LIN {X 0,Y 526.698,Z 428.469,A -85,B 0,C 180,E1 -4749.903,E2 -4749.903} C_VEL
LIN {X 0,Y 526.188,Z 442.456,A -85,B 0,C 180,E1 -4750.797,E2 -4750.797} C_VEL
LIN {X 0,Y 525.617,Z 456.418,A -85,B 0,C 180,E1 -4751.866,E2 -4751.866} C_VEL
LIN {X 0,Y 525.179,Z 468.801,A -85,B 0,C 180,E1 -4752.978,E2 -4752.978} C_VEL
LIN {X 0,Y 524.752,Z 481.132,A -85,B 0,C 180,E1 -4754.263,E2 -4754.263} C_VEL
LIN {X 0,Y 524.384,Z 492.437,A -85,B 0,C 180,E1 -4755.644,E2 -4755.644} C_VEL
LIN {X 0,Y 524.046,Z 503.255,A -85,B 0,C 180,E1 -4757.215,E2 -4757.215} C_VEL
LIN {X 0,Y 523.793,Z 512.276,A -85,B 0,C 180,E1 -4758.781,E2 -4758.781} C_VEL
LIN {X 0,Y 523.564,Z 519.801,A -85,B 0,C 180,E1 -4760.34,E2 -4760.34} C_VEL
LIN {X 0,Y 523.503,Z 526.021,A -85,B 0,C 180,E1 -4761.896,E2 -4761.896} C_VEL
LIN {X 0,Y 523.45,Z 531.029,A -85,B 0,C 180,E1 -4763.485,E2 -4763.485} C_VEL
LIN {X 0,Y 523.398,Z 533.892,A -85,B 0,C 180,E1 -4764.606,E2 -4764.606} C_VEL
LIN {X 0,Y 523.38,Z 536.906,A -85,B 0,C 180,E1 -4766.15,E2 -4766.15} C_VEL
LIN {X 0,Y 523.33,Z 538.868,A -85,B 0,C 180,E1 -4767.691,E2 -4767.691} C_VEL
LIN {X 0,Y 523.247,Z 539.833,A -85,B 0,C 180,E1 -4769.23,E2 -4769.23} C_VEL
LIN {X 0,Y 523.247,Z 539.832,A -85,B 0,C 180,E1 -4770.769,E2 -4770.769} C_VEL
LIN {X 0,Y 523.33,Z 538.868,A -85,B 0,C 180,E1 -4772.308,E2 -4772.308} C_VEL
LIN {X 0,Y 523.38,Z 536.906,A -85,B 0,C 180,E1 -4773.849,E2 -4773.849} C_VEL
LIN {X 0,Y 523.397,Z 533.906,A -85,B 0,C 180,E1 -4775.393,E2 -4775.393} C_VEL
LIN {X 0,Y 523.457,Z 529.853,A -85,B 0,C 180,E1 -4776.94,E2 -4776.94} C_VEL
LIN {X 0,Y 523.523,Z 524.622,A -85,B 0,C 180,E1 -4778.491,E2 -4778.491} C_VEL
LIN {X 0,Y 523.624,Z 518.224,A -85,B 0,C 180,E1 -4780.048,E2 -4780.048} C_VEL
LIN {X 0,Y 523.883,Z 510.045,A -85,B 0,C 180,E1 -4781.676,E2 -4781.676} C_VEL
LIN {X 0,Y 524.093,Z 501.032,A -85,B 0,C 180,E1 -4783.177,E2 -4783.177} C_VEL
LIN {X 0,Y 524.474,Z 491.393,A -85,B 0,C 180,E1 -4784.551,E2 -4784.551} C_VEL
LIN {X 0,Y 524.874,Z 480.123,A -85,B 0,C 180,E1 -4785.931,E2 -4785.931} C_VEL
LIN {X 0,Y 525.428,Z 466.759,A -85,B 0,C 180,E1 -4787.314,E2 -4787.314} C_VEL
LIN {X 0,Y 525.923,Z 454.174,A -85,B 0,C 180,E1 -4788.417,E2 -4788.417} C_VEL
LIN {X 0,Y 526.459,Z 439.758,A -85,B 0,C 180,E1 -4789.495,E2 -4789.495} C_VEL
LIN {X 0,Y 527.012,Z 425.551,A -85,B 0,C 180,E1 -4790.388,E2 -4790.388} C_VEL
LIN {X 0,Y 527.61,Z 410.217,A -85,B 0,C 180,E1 -4791.184,E2 -4791.184} C_VEL
LIN {X 0,Y 528.07,Z 394.743,A -85,B 0,C 180,E1 -4791.822,E2 -4791.822} C_VEL
LIN {X 0,Y 528.514,Z 378.995,A -85,B 0,C 180,E1 -4792.322,E2 -4792.322} C_VEL
LIN {X 0,Y 528.836,Z 362.769,A -85,B 0,C 180,E1 -4792.694,E2 -4792.694} C_VEL
LIN {X 0,Y 529.26,Z 309.626,A -85,B 0,C 180,E1 -4793.476,E2 -4793.476} C_VEL
LIN {X 0,Y 530.388,Z 201.86,A -85,B 0,C 180,E1 -4795.062,E2 -4795.062} C_VEL
LIN {X 0,Y 530.606,Z 171.21,A -85,B 0,C 180,E1 -4795.535,E2 -4795.535} C_VEL
LIN {X 0,Y 528.283,Z 155.627,A -85,B 0,C 180,E1 -4795.933,E2 -4795.933} C_VEL
LIN {X 0,Y 529.372,Z 120.749,A -85,B 0,C 180,E1 -4798.908,E2 -4798.908} C_VEL
LIN {X 0,Y 529.593,Z 109.375,A -85,B 0,C 180,E1 -4799.898,E2 -4799.898} C_VEL
LIN {X 0,Y 523.945,Z 91.535,A -85,B 0,C 180,E1 -4801.852,E2 -4801.852} C_VEL
LIN {X 0,Y 523.935,Z 91.535,A -85,B 0,C 180,E1 -4804.289,E2 -4804.289} C_VEL
LIN {X 0,Y 523.903,Z 91.537,A -85,B 0,C 180,E1 -4807.132,E2 -4807.132} C_VEL
LIN {X 0,Y 523.933,Z 91.535,A -85,B 0,C 180,E1 -4810.129,E2 -4810.129} C_VEL
LIN {X 0,Y 523.935,Z 91.538,A -85,B 0,C 180,E1 -4812.459,E2 -4812.459} C_VEL
LIN {X 0,Y 523.951,Z 91.528,A -85,B 0,C 180,E1 -4815.308,E2 -4815.308} C_VEL
LIN {X 0,Y 523.954,Z 91.53,A -85,B 0,C 180,E1 -4818.689,E2 -4818.689} C_VEL
LIN {X 0,Y 523.913,Z 91.535,A -85,B 0,C 180,E1 -4821.898,E2 -4821.898} C_VEL
LIN {X 0,Y 523.934,Z 91.53,A -85,B 0,C 180,E1 -4824.909,E2 -4824.909} C_VEL
LIN {X 0,Y 523.934,Z 91.531,A -85,B 0,C 180,E1 -4827.679,E2 -4827.679} C_VEL
LIN {X 0,Y 523.956,Z 91.528,A -85,B 0,C 180,E1 -4830.675,E2 -4830.675} C_VEL
LIN {X 0,Y 523.97,Z 91.528,A -85,B 0,C 180,E1 -4833.728,E2 -4833.728} C_VEL
LIN {X 0,Y 523.932,Z 91.535,A -85,B 0,C 180,E1 -4836.271,E2 -4836.271} C_VEL
LIN {X 0,Y 523.941,Z 91.528,A -85,B 0,C 180,E1 -4838.767,E2 -4838.767} C_VEL
LIN {X 0,Y 523.948,Z 91.528,A -85,B 0,C 180,E1 -4841.221,E2 -4841.221} C_VEL
LIN {X 0,Y 523.933,Z 91.534,A -85,B 0,C 180,E1 -4843.639,E2 -4843.639} C_VEL
LIN {X 0,Y 523.937,Z 91.535,A -85,B 0,C 180,E1 -4846.028,E2 -4846.028} C_VEL
LIN {X 0,Y 524.01,Z 91.521,A -85,B 0,C 180,E1 -4848.394,E2 -4848.394} C_VEL
LIN {X 0,Y 523.999,Z 91.526,A -85,B 0,C 180,E1 -4851.516,E2 -4851.516} C_VEL
LIN {X 0,Y 524.078,Z 91.511,A -85,B 0,C 180,E1 -4854.614,E2 -4854.614} C_VEL
LIN {X 0,Y 524.107,Z 91.516,A -85,B 0,C 180,E1 -4857.695,E2 -4857.695} C_VEL
LIN {X 0,Y 524.119,Z 91.506,A -85,B 0,C 180,E1 -4860.768,E2 -4860.768} C_VEL
LIN {X 0,Y 524.069,Z 91.514,A -85,B 0,C 180,E1 -4863.075,E2 -4863.075} C_VEL
LIN {X 0,Y 524.042,Z 91.517,A -85,B 0,C 180,E1 -4866.159,E2 -4866.159} C_VEL
LIN {X 0,Y 523.993,Z 91.527,A -85,B 0,C 180,E1 -4869.262,E2 -4869.262} C_VEL
LIN {X 0,Y 523.999,Z 91.525,A -85,B 0,C 180,E1 -4871.74,E2 -4871.74} C_VEL
LIN {X 0,Y 523.989,Z 91.526,A -85,B 0,C 180,E1 -4875.053,E2 -4875.053} C_VEL
LIN {X 0,Y 523.96,Z 91.527,A -85,B 0,C 180,E1 -4877.969,E2 -4877.969} C_VEL
LIN {X 0,Y 523.968,Z 91.525,A -85,B 0,C 180,E1 -4880.41,E2 -4880.41} C_VEL
LIN {X 0,Y 523.913,Z 91.536,A -85,B 0,C 180,E1 -4882.893,E2 -4882.893} C_VEL
LIN {X 0,Y 523.949,Z 91.532,A -85,B 0,C 180,E1 -4885.419,E2 -4885.419} C_VEL
LIN {X 0,Y 523.965,Z 91.525,A -85,B 0,C 180,E1 -4887.999,E2 -4887.999} C_VEL
LIN {X 0,Y 523.943,Z 91.533,A -85,B 0,C 180,E1 -4890.856,E2 -4890.856} C_VEL
LIN {X 0,Y 523.958,Z 91.527,A -85,B 0,C 180,E1 -4893.735,E2 -4893.735} C_VEL
LIN {X 0,Y 523.919,Z 91.532,A -85,B 0,C 180,E1 -4896.405,E2 -4896.405} C_VEL
LIN {X 0,Y 523.921,Z 91.537,A -85,B 0,C 180,E1 -4899.085,E2 -4899.085} C_VEL
LIN {X 0,Y 523.953,Z 91.527,A -85,B 0,C 180,E1 -4902.119,E2 -4902.119} C_VEL
LIN {X 0,Y 523.953,Z 91.529,A -85,B 0,C 180,E1 -4905.309,E2 -4905.309} C_VEL
LIN {X 0,Y 523.92,Z 91.538,A -85,B 0,C 180,E1 -4906.914,E2 -4906.914} C_VEL
LIN {X 0,Y 523.253,Z 91.616,A -85,B 0,C 180,E1 -4907.555,E2 -4907.555} C_VEL
LIN {X 0,Y 520.408,Z 91.974,A -85,B 0,C 180,E1 -4908.597,E2 -4908.597} C_VEL
LIN {X 0,Y 518.002,Z 92.271,A -85,B 0,C 180,E1 -4909.436,E2 -4909.436} C_VEL
LIN {X 0,Y 516.965,Z 92.399,A -85,B 0,C 180,E1 -4910.083,E2 -4910.083} C_VEL
LIN {X 0,Y 516.879,Z 92.41,A -85,B 0,C 180,E1 -4910.303,E2 -4910.303} C_VEL
LIN {X 0,Y 516.874,Z 92.409,A -85,B 0,C 180,E1 -4913.344,E2 -4913.344} C_VEL
LIN {X 0,Y 516.905,Z 92.406,A -85,B 0,C 180,E1 -4916.121,E2 -4916.121} C_VEL
LIN {X 0,Y 516.889,Z 92.411,A -85,B 0,C 180,E1 -4918.936,E2 -4918.936} C_VEL
LIN {X 0,Y 516.917,Z 92.403,A -85,B 0,C 180,E1 -4921.585,E2 -4921.585} C_VEL
LIN {X 0,Y 516.93,Z 92.406,A -85,B 0,C 180,E1 -4924.212,E2 -4924.212} C_VEL
LIN {X 0,Y 516.87,Z 92.413,A -85,B 0,C 180,E1 -4926.777,E2 -4926.777} C_VEL
LIN {X 0,Y 516.938,Z 92.401,A -85,B 0,C 180,E1 -4929.732,E2 -4929.732} C_VEL
LIN {X 0,Y 516.928,Z 92.407,A -85,B 0,C 180,E1 -4932.597,E2 -4932.597} C_VEL
LIN {X 0,Y 516.942,Z 92.401,A -85,B 0,C 180,E1 -4935.031,E2 -4935.031} C_VEL
LIN {X 0,Y 516.966,Z 92.406,A -85,B 0,C 180,E1 -4938.234,E2 -4938.234} C_VEL
LIN {X 0,Y 516.968,Z 92.397,A -85,B 0,C 180,E1 -4941.4,E2 -4941.4} C_VEL
LIN {X 0,Y 517.011,Z 92.395,A -85,B 0,C 180,E1 -4943.757,E2 -4943.757} C_VEL
LIN {X 0,Y 517.085,Z 92.385,A -85,B 0,C 180,E1 -4947.664,E2 -4947.664} C_VEL
LIN {X 0,Y 517.094,Z 92.382,A -85,B 0,C 180,E1 -4950.779,E2 -4950.779} C_VEL
LIN {X 0,Y 517.012,Z 92.391,A -85,B 0,C 180,E1 -4953.117,E2 -4953.117} C_VEL
LIN {X 0,Y 517.011,Z 92.396,A -85,B 0,C 180,E1 -4956.244,E2 -4956.244} C_VEL
LIN {X 0,Y 516.953,Z 92.401,A -85,B 0,C 180,E1 -4959.39,E2 -4959.39} C_VEL
LIN {X 0,Y 516.954,Z 92.407,A -85,B 0,C 180,E1 -4961.808,E2 -4961.808} C_VEL
LIN {X 0,Y 516.946,Z 92.4,A -85,B 0,C 180,E1 -4965.147,E2 -4965.147} C_VEL
LIN {X 0,Y 516.927,Z 92.404,A -85,B 0,C 180,E1 -4968.223,E2 -4968.223} C_VEL
LIN {X 0,Y 516.915,Z 92.403,A -85,B 0,C 180,E1 -4970.702,E2 -4970.702} C_VEL
LIN {X 0,Y 516.894,Z 92.409,A -85,B 0,C 180,E1 -4974.073,E2 -4974.073} C_VEL
LIN {X 0,Y 516.928,Z 92.402,A -85,B 0,C 180,E1 -4976.658,E2 -4976.658} C_VEL
LIN {X 0,Y 516.913,Z 92.412,A -85,B 0,C 180,E1 -4979.524,E2 -4979.524} C_VEL
LIN {X 0,Y 516.9,Z 92.405,A -85,B 0,C 180,E1 -4982.544,E2 -4982.544} C_VEL
LIN {X 0,Y 516.869,Z 92.416,A -85,B 0,C 180,E1 -4985.33,E2 -4985.33} C_VEL
LIN {X 0,Y 516.882,Z 92.409,A -85,B 0,C 180,E1 -4987.943,E2 -4987.943} C_VEL
LIN {X 0,Y 516.886,Z 92.408,A -85,B 0,C 180,E1 -4990.742,E2 -4990.742} C_VEL
LIN {X 0,Y 516.886,Z 92.409,A -85,B 0,C 180,E1 -4992.832,E2 -4992.832} C_VEL
LIN {X 0,Y 516.926,Z 92.407,A -85,B 0,C 180,E1 -4995.01,E2 -4995.01} C_VEL
LIN {X 0,Y 516.916,Z 92.403,A -85,B 0,C 180,E1 -4998.399,E2 -4998.399} C_VEL
LIN {X 0,Y 516.884,Z 92.414,A -85,B 0,C 180,E1 -5001.284,E2 -5001.284} C_VEL
LIN {X 0,Y 516.88,Z 92.409,A -85,B 0,C 180,E1 -5004.22,E2 -5004.22} C_VEL
LIN {X 0,Y 516.898,Z 92.414,A -85,B 0,C 180,E1 -5007.053,E2 -5007.053} C_VEL
LIN {X 0,Y 516.896,Z 92.409,A -85,B 0,C 180,E1 -5009.797,E2 -5009.797} C_VEL
LIN {X 0,Y 516.93,Z 92.408,A -85,B 0,C 180,E1 -5012.467,E2 -5012.467} C_VEL
LIN {X 0,Y 516.94,Z 92.407,A -85,B 0,C 180,E1 -5013.709,E2 -5013.709} C_VEL
LIN {X 0,Y 517.988,Z 95.336,A -85,B 0,C 180,E1 -5013.83,E2 -5013.83} C_VEL
LIN {X 0,Y 524.276,Z 108.483,A -85,B 0,C 180,E1 -5014.383,E2 -5014.383} C_VEL
LIN {X 0,Y 522.69,Z 254.21,A -85,B 0,C 180,E1 -5016.605,E2 -5016.605} C_VEL
LIN {X 0,Y 522.29,Z 290.172,A -85,B 0,C 180,E1 -5017.162,E2 -5017.162} C_VEL
LIN {X 0,Y 521.965,Z 307.306,A -85,B 0,C 180,E1 -5017.591,E2 -5017.591} C_VEL
LIN {X 0,Y 521.509,Z 323.109,A -85,B 0,C 180,E1 -5018.144,E2 -5018.144} C_VEL
LIN {X 0,Y 521.037,Z 338.718,A -85,B 0,C 180,E1 -5018.85,E2 -5018.85} C_VEL
LIN {X 0,Y 520.492,Z 353.18,A -85,B 0,C 180,E1 -5019.654,E2 -5019.654} C_VEL
LIN {X 0,Y 519.849,Z 368.084,A -85,B 0,C 180,E1 -5020.657,E2 -5020.657} C_VEL
LIN {X 0,Y 519.233,Z 381.509,A -85,B 0,C 180,E1 -5021.744,E2 -5021.744} C_VEL
LIN {X 0,Y 518.651,Z 393.241,A -85,B 0,C 180,E1 -5022.859,E2 -5022.859} C_VEL
LIN {X 0,Y 518.193,Z 404.191,A -85,B 0,C 180,E1 -5024.059,E2 -5024.059} C_VEL
LIN {X 0,Y 517.695,Z 415.067,A -85,B 0,C 180,E1 -5025.455,E2 -5025.455} C_VEL
LIN {X 0,Y 517.26,Z 425.524,A -85,B 0,C 180,E1 -5027.045,E2 -5027.045} C_VEL
LIN {X 0,Y 516.92,Z 434.225,A -85,B 0,C 180,E1 -5028.63,E2 -5028.63} C_VEL
LIN {X 0,Y 516.636,Z 441.519,A -85,B 0,C 180,E1 -5030.21,E2 -5030.21} C_VEL
LIN {X 0,Y 516.517,Z 447.491,A -85,B 0,C 180,E1 -5031.786,E2 -5031.786} C_VEL
LIN {X 0,Y 516.437,Z 452.437,A -85,B 0,C 180,E1 -5033.431,E2 -5033.431} C_VEL
LIN {X 0,Y 516.334,Z 455.124,A -85,B 0,C 180,E1 -5034.533,E2 -5034.533} C_VEL
LIN {X 0,Y 516.327,Z 458.021,A -85,B 0,C 180,E1 -5036.097,E2 -5036.097} C_VEL
LIN {X 0,Y 516.255,Z 459.965,A -85,B 0,C 180,E1 -5037.659,E2 -5037.659} C_VEL
LIN {X 0,Y 516.186,Z 460.93,A -85,B 0,C 180,E1 -5039.22,E2 -5039.22} C_VEL
LIN {X 0,Y 516.189,Z 460.981,A -85,B 0,C 180,E1 -5040.78,E2 -5040.78} C_VEL
LIN {X 0,Y 516.257,Z 460.095,A -85,B 0,C 180,E1 -5042.341,E2 -5042.341} C_VEL
LIN {X 0,Y 516.341,Z 458.242,A -85,B 0,C 180,E1 -5043.902,E2 -5043.902} C_VEL
LIN {X 0,Y 516.338,Z 455.456,A -85,B 0,C 180,E1 -5045.467,E2 -5045.467} C_VEL
LIN {X 0,Y 516.476,Z 451.597,A -85,B 0,C 180,E1 -5047.034,E2 -5047.034} C_VEL
LIN {X 0,Y 516.525,Z 446.628,A -85,B 0,C 180,E1 -5048.608,E2 -5048.608} C_VEL
LIN {X 0,Y 516.701,Z 440.491,A -85,B 0,C 180,E1 -5050.185,E2 -5050.185} C_VEL
LIN {X 0,Y 516.99,Z 432.998,A -85,B 0,C 180,E1 -5051.766,E2 -5051.766} C_VEL
LIN {X 0,Y 517.368,Z 423.951,A -85,B 0,C 180,E1 -5053.352,E2 -5053.352} C_VEL
LIN {X 0,Y 517.764,Z 414.573,A -85,B 0,C 180,E1 -5054.744,E2 -5054.744} C_VEL
LIN {X 0,Y 518.272,Z 403.549,A -85,B 0,C 180,E1 -5056.14,E2 -5056.14} C_VEL
LIN {X 0,Y 518.798,Z 391.418,A -85,B 0,C 180,E1 -5057.441,E2 -5057.441} C_VEL
LIN {X 0,Y 519.406,Z 378.461,A -85,B 0,C 180,E1 -5058.61,E2 -5058.61} C_VEL
LIN {X 0,Y 519.915,Z 364.877,A -85,B 0,C 180,E1 -5059.648,E2 -5059.648} C_VEL
LIN {X 0,Y 520.439,Z 350.731,A -85,B 0,C 180,E1 -5060.555,E2 -5060.555} C_VEL
LIN {X 0,Y 521.023,Z 335.381,A -85,B 0,C 180,E1 -5061.358,E2 -5061.358} C_VEL
LIN {X 0,Y 521.419,Z 319.929,A -85,B 0,C 180,E1 -5062.001,E2 -5062.001} C_VEL
LIN {X 0,Y 521.748,Z 303.332,A -85,B 0,C 180,E1 -5062.523,E2 -5062.523} C_VEL
LIN {X 0,Y 521.951,Z 287.036,A -85,B 0,C 180,E1 -5062.88,E2 -5062.88} C_VEL
LIN {X 0,Y 523.479,Z 165.935,A -85,B 0,C 180,E1 -5064.773,E2 -5064.773} C_VEL
LIN {X 0,Y 524.468,Z 108.668,A -85,B 0,C 180,E1 -5065.737,E2 -5065.737} C_VEL
LIN {X 0,Y 518.182,Z 95.78,A -85,B 0,C 180,E1 -5066.361,E2 -5066.361} C_VEL
LIN {X 0,Y 516.963,Z 93.096,A -85,B 0,C 180,E1 -5066.487,E2 -5066.487} C_VEL
LIN {X 0,Y 516.837,Z 92.42,A -85,B 0,C 180,E1 -5066.521,E2 -5066.521} C_VEL
LIN {X 0,Y 516.881,Z 92.414,A -85,B 0,C 180,E1 -5069.517,E2 -5069.517} C_VEL
LIN {X 0,Y 516.893,Z 92.415,A -85,B 0,C 180,E1 -5072.542,E2 -5072.542} C_VEL
LIN {X 0,Y 516.865,Z 92.414,A -85,B 0,C 180,E1 -5075.329,E2 -5075.329} C_VEL
LIN {X 0,Y 516.879,Z 92.414,A -85,B 0,C 180,E1 -5077.942,E2 -5077.942} C_VEL
LIN {X 0,Y 516.884,Z 92.413,A -85,B 0,C 180,E1 -5080.741,E2 -5080.741} C_VEL
LIN {X 0,Y 516.884,Z 92.412,A -85,B 0,C 180,E1 -5082.831,E2 -5082.831} C_VEL
LIN {X 0,Y 516.897,Z 92.409,A -85,B 0,C 180,E1 -5085.007,E2 -5085.007} C_VEL
LIN {X 0,Y 516.915,Z 92.41,A -85,B 0,C 180,E1 -5088.398,E2 -5088.398} C_VEL
LIN {X 0,Y 516.882,Z 92.414,A -85,B 0,C 180,E1 -5091.284,E2 -5091.284} C_VEL
LIN {X 0,Y 516.872,Z 92.417,A -85,B 0,C 180,E1 -5094.219,E2 -5094.219} C_VEL
LIN {X 0,Y 516.897,Z 92.418,A -85,B 0,C 180,E1 -5097.053,E2 -5097.053} C_VEL
LIN {X 0,Y 516.957,Z 92.588,A -85,B 0,C 180,E1 -5097.98,E2 -5097.98} C_VEL
LIN {X 0,Y 521.725,Z 108.054,A -85,B 0,C 180,E1 -5099.788,E2 -5099.788} C_VEL
LIN {X 0,Y 522.518,Z 111.509,A -85,B 0,C 180,E1 -5100.154,E2 -5100.154} C_VEL
LIN {X 0,Y 521.372,Z 141.954,A -85,B 0,C 180,E1 -5102.831,E2 -5102.831} C_VEL
LIN {X 0,Y 521.076,Z 151.687,A -85,B 0,C 180,E1 -5103.668,E2 -5103.668} C_VEL
LIN {X 0,Y 524.053,Z 173.701,A -85,B 0,C 180,E1 -5104.228,E2 -5104.228} C_VEL
LIN {X 0,Y 522.395,Z 292.457,A -85,B 0,C 180,E1 -5106.117,E2 -5106.117} C_VEL
LIN {X 0,Y 521.708,Z 362.986,A -85,B 0,C 180,E1 -5107.187,E2 -5107.187} C_VEL
LIN {X 0,Y 521.337,Z 380.565,A -85,B 0,C 180,E1 -5107.614,E2 -5107.614} C_VEL
LIN {X 0,Y 520.88,Z 396.793,A -85,B 0,C 180,E1 -5108.167,E2 -5108.167} C_VEL
LIN {X 0,Y 520.346,Z 412.264,A -85,B 0,C 180,E1 -5108.842,E2 -5108.842} C_VEL
LIN {X 0,Y 519.81,Z 426.912,A -85,B 0,C 180,E1 -5109.625,E2 -5109.625} C_VEL
LIN {X 0,Y 519.269,Z 441.013,A -85,B 0,C 180,E1 -5110.531,E2 -5110.531} C_VEL
LIN {X 0,Y 518.675,Z 455.327,A -85,B 0,C 180,E1 -5111.63,E2 -5111.63} C_VEL
LIN {X 0,Y 518.168,Z 468.684,A -85,B 0,C 180,E1 -5112.842,E2 -5112.842} C_VEL
LIN {X 0,Y 517.762,Z 480.106,A -85,B 0,C 180,E1 -5114.045,E2 -5114.045} C_VEL
LIN {X 0,Y 517.368,Z 491.488,A -85,B 0,C 180,E1 -5115.445,E2 -5115.445} C_VEL
LIN {X 0,Y 516.952,Z 502.384,A -85,B 0,C 180,E1 -5117.037,E2 -5117.037} C_VEL
LIN {X 0,Y 516.79,Z 509.654,A -85,B 0,C 180,E1 -5118.279,E2 -5118.279} C_VEL
LIN {X 0,Y 516.559,Z 517.352,A -85,B 0,C 180,E1 -5119.812,E2 -5119.812} C_VEL
LIN {X 0,Y 516.453,Z 523.852,A -85,B 0,C 180,E1 -5121.391,E2 -5121.391} C_VEL
LIN {X 0,Y 516.377,Z 529.177,A -85,B 0,C 180,E1 -5122.964,E2 -5122.964} C_VEL
LIN {X 0,Y 516.327,Z 533.277,A -85,B 0,C 180,E1 -5124.532,E2 -5124.532} C_VEL
LIN {X 0,Y 516.305,Z 536.329,A -85,B 0,C 180,E1 -5126.097,E2 -5126.097} C_VEL
LIN {X 0,Y 516.256,Z 538.32,A -85,B 0,C 180,E1 -5127.659,E2 -5127.659} C_VEL
LIN {X 0,Y 516.166,Z 539.314,A -85,B 0,C 180,E1 -5129.219,E2 -5129.219} C_VEL
LIN {X 0,Y 516.166,Z 539.319,A -85,B 0,C 180,E1 -5130.78,E2 -5130.78} C_VEL
LIN {X 0,Y 516.256,Z 538.349,A -85,B 0,C 180,E1 -5132.34,E2 -5132.34} C_VEL
LIN {X 0,Y 516.305,Z 536.374,A -85,B 0,C 180,E1 -5133.902,E2 -5133.902} C_VEL
LIN {X 0,Y 516.326,Z 533.364,A -85,B 0,C 180,E1 -5135.467,E2 -5135.467} C_VEL
LIN {X 0,Y 516.376,Z 529.3,A -85,B 0,C 180,E1 -5137.035,E2 -5137.035} C_VEL
LIN {X 0,Y 516.455,Z 524.047,A -85,B 0,C 180,E1 -5138.608,E2 -5138.608} C_VEL
LIN {X 0,Y 516.561,Z 517.619,A -85,B 0,C 180,E1 -5140.187,E2 -5140.187} C_VEL
LIN {X 0,Y 516.801,Z 509.778,A -85,B 0,C 180,E1 -5141.77,E2 -5141.77} C_VEL
LIN {X 0,Y 517.091,Z 500.371,A -85,B 0,C 180,E1 -5143.359,E2 -5143.359} C_VEL
LIN {X 0,Y 517.464,Z 489.152,A -85,B 0,C 180,E1 -5144.954,E2 -5144.954} C_VEL
LIN {X 0,Y 517.952,Z 477.535,A -85,B 0,C 180,E1 -5146.352,E2 -5146.352} C_VEL
LIN {X 0,Y 518.521,Z 464.876,A -85,B 0,C 180,E1 -5147.653,E2 -5147.653} C_VEL
LIN {X 0,Y 519.066,Z 451.613,A -85,B 0,C 180,E1 -5148.814,E2 -5148.814} C_VEL
LIN {X 0,Y 519.692,Z 437.359,A -85,B 0,C 180,E1 -5149.863,E2 -5149.863} C_VEL
LIN {X 0,Y 520.307,Z 422.946,A -85,B 0,C 180,E1 -5150.752,E2 -5150.752} C_VEL
LIN {X 0,Y 520.9,Z 407.287,A -85,B 0,C 180,E1 -5151.55,E2 -5151.55} C_VEL
LIN {X 0,Y 521.448,Z 392.036,A -85,B 0,C 180,E1 -5152.171,E2 -5152.171} C_VEL
LIN {X 0,Y 521.856,Z 375.621,A -85,B 0,C 180,E1 -5152.674,E2 -5152.674} C_VEL
LIN {X 0,Y 522.216,Z 359.174,A -85,B 0,C 180,E1 -5153.022,E2 -5153.022} C_VEL
LIN {X 0,Y 523.526,Z 237.483,A -85,B 0,C 180,E1 -5154.856,E2 -5154.856} C_VEL
LIN {X 0,Y 524.19,Z 172.24,A -85,B 0,C 180,E1 -5155.847,E2 -5155.847} C_VEL
LIN {X 0,Y 521.619,Z 155.534,A -85,B 0,C 180,E1 -5156.263,E2 -5156.263} C_VEL
LIN {X 0,Y 522.793,Z 121.957,A -85,B 0,C 180,E1 -5159.163,E2 -5159.163} C_VEL
LIN {X 0,Y 523.145,Z 112.783,A -85,B 0,C 180,E1 -5159.964,E2 -5159.964} C_VEL
LIN {X 0,Y 519.785,Z 101.473,A -85,B 0,C 180,E1 -5161.186,E2 -5161.186} C_VEL
LIN {X 0,Y 516.919,Z 92.411,A -85,B 0,C 180,E1 -5162.201,E2 -5162.201} C_VEL
LIN {X 0,Y 516.883,Z 92.415,A -85,B 0,C 180,E1 -5164.824,E2 -5164.824} C_VEL
LIN {X 0,Y 516.876,Z 92.412,A -85,B 0,C 180,E1 -5167.943,E2 -5167.943} C_VEL
LIN {X 0,Y 516.88,Z 92.415,A -85,B 0,C 180,E1 -5170.741,E2 -5170.741} C_VEL
LIN {X 0,Y 516.9,Z 92.41,A -85,B 0,C 180,E1 -5172.829,E2 -5172.829} C_VEL
LIN {X 0,Y 516.918,Z 92.406,A -85,B 0,C 180,E1 -5175.01,E2 -5175.01} C_VEL
LIN {X 0,Y 516.91,Z 92.412,A -85,B 0,C 180,E1 -5178.398,E2 -5178.398} C_VEL
LIN {X 0,Y 516.879,Z 92.408,A -85,B 0,C 180,E1 -5181.284,E2 -5181.284} C_VEL
LIN {X 0,Y 516.886,Z 92.416,A -85,B 0,C 180,E1 -5184.221,E2 -5184.221} C_VEL
LIN {X 0,Y 516.892,Z 92.406,A -85,B 0,C 180,E1 -5187.053,E2 -5187.053} C_VEL
LIN {X 0,Y 516.895,Z 92.409,A -85,B 0,C 180,E1 -5189.797,E2 -5189.797} C_VEL
LIN {X 0,Y 516.923,Z 92.406,A -85,B 0,C 180,E1 -5192.467,E2 -5192.467} C_VEL
LIN {X 0,Y 516.906,Z 92.404,A -85,B 0,C 180,E1 -5195.072,E2 -5195.072} C_VEL
LIN {X 0,Y 516.865,Z 92.413,A -85,B 0,C 180,E1 -5197.622,E2 -5197.622} C_VEL
LIN {X 0,Y 516.928,Z 92.408,A -85,B 0,C 180,E1 -5200.13,E2 -5200.13} C_VEL
LIN {X 0,Y 516.925,Z 92.403,A -85,B 0,C 180,E1 -5202.596,E2 -5202.596} C_VEL
LIN {X 0,Y 516.938,Z 92.4,A -85,B 0,C 180,E1 -5205.03,E2 -5205.03} C_VEL
LIN {X 0,Y 517,Z 92.396,A -85,B 0,C 180,E1 -5208.235,E2 -5208.235} C_VEL
LIN {X 0,Y 516.964,Z 92.401,A -85,B 0,C 180,E1 -5211.4,E2 -5211.4} C_VEL
LIN {X 0,Y 517.006,Z 92.401,A -85,B 0,C 180,E1 -5213.757,E2 -5213.757} C_VEL
LIN {X 0,Y 517.079,Z 92.392,A -85,B 0,C 180,E1 -5217.663,E2 -5217.663} C_VEL
LIN {X 0,Y 517.089,Z 92.382,A -85,B 0,C 180,E1 -5220.779,E2 -5220.779} C_VEL
LIN {X 0,Y 517.01,Z 92.394,A -85,B 0,C 180,E1 -5223.117,E2 -5223.117} C_VEL
LIN {X 0,Y 517.006,Z 92.393,A -85,B 0,C 180,E1 -5226.243,E2 -5226.243} C_VEL
LIN {X 0,Y 516.947,Z 92.407,A -85,B 0,C 180,E1 -5229.389,E2 -5229.389} C_VEL
LIN {X 0,Y 516.948,Z 92.403,A -85,B 0,C 180,E1 -5231.807,E2 -5231.807} C_VEL
LIN {X 0,Y 516.94,Z 92.406,A -85,B 0,C 180,E1 -5235.147,E2 -5235.147} C_VEL
LIN {X 0,Y 516.922,Z 92.402,A -85,B 0,C 180,E1 -5238.222,E2 -5238.222} C_VEL
LIN {X 0,Y 516.908,Z 92.406,A -85,B 0,C 180,E1 -5240.702,E2 -5240.702} C_VEL
LIN {X 0,Y 516.908,Z 92.404,A -85,B 0,C 180,E1 -5244.072,E2 -5244.072} C_VEL
LIN {X 0,Y 516.922,Z 92.405,A -85,B 0,C 180,E1 -5246.658,E2 -5246.658} C_VEL
LIN {X 0,Y 516.907,Z 92.407,A -85,B 0,C 180,E1 -5249.524,E2 -5249.524} C_VEL
LIN {X 0,Y 516.897,Z 92.408,A -85,B 0,C 180,E1 -5252.545,E2 -5252.545} C_VEL
LIN {X 0,Y 516.879,Z 92.412,A -85,B 0,C 180,E1 -5255.333,E2 -5255.333} C_VEL
LIN {X 0,Y 516.878,Z 92.408,A -85,B 0,C 180,E1 -5257.944,E2 -5257.944} C_VEL
LIN {X 0,Y 516.882,Z 92.414,A -85,B 0,C 180,E1 -5260.742,E2 -5260.742} C_VEL
LIN {X 0,Y 516.9,Z 92.413,A -85,B 0,C 180,E1 -5262.83,E2 -5262.83} C_VEL
LIN {X 0,Y 516.919,Z 92.409,A -85,B 0,C 180,E1 -5265.011,E2 -5265.011} C_VEL
LIN {X 0,Y 516.915,Z 92.407,A -85,B 0,C 180,E1 -5268.399,E2 -5268.399} C_VEL
LIN {X 0,Y 516.879,Z 92.41,A -85,B 0,C 180,E1 -5270.303,E2 -5270.303} C_VEL
LIN {X 0,Y 516.209,Z 92.499,A -85,B 0,C 180,E1 -5270.953,E2 -5270.953} C_VEL
LIN {X 0,Y 513.362,Z 92.85,A -85,B 0,C 180,E1 -5272.008,E2 -5272.008} C_VEL
LIN {X 0,Y 510.951,Z 93.153,A -85,B 0,C 180,E1 -5272.859,E2 -5272.859} C_VEL
LIN {X 0,Y 509.907,Z 93.277,A -85,B 0,C 180,E1 -5273.515,E2 -5273.515} C_VEL
LIN {X 0,Y 509.817,Z 93.287,A -85,B 0,C 180,E1 -5273.738,E2 -5273.738} C_VEL
LIN {X 0,Y 509.857,Z 93.29,A -85,B 0,C 180,E1 -5276.54,E2 -5276.54} C_VEL
LIN {X 0,Y 509.843,Z 93.285,A -85,B 0,C 180,E1 -5279.335,E2 -5279.335} C_VEL
LIN {X 0,Y 509.892,Z 93.28,A -85,B 0,C 180,E1 -5282.055,E2 -5282.055} C_VEL
LIN {X 0,Y 509.876,Z 93.286,A -85,B 0,C 180,E1 -5284.705,E2 -5284.705} C_VEL
LIN {X 0,Y 509.826,Z 93.286,A -85,B 0,C 180,E1 -5287.458,E2 -5287.458} C_VEL
LIN {X 0,Y 509.916,Z 93.277,A -85,B 0,C 180,E1 -5289.845,E2 -5289.845} C_VEL
LIN {X 0,Y 509.883,Z 93.279,A -85,B 0,C 180,E1 -5293.175,E2 -5293.175} C_VEL
LIN {X 0,Y 509.864,Z 93.283,A -85,B 0,C 180,E1 -5295.635,E2 -5295.635} C_VEL
LIN {X 0,Y 509.913,Z 93.277,A -85,B 0,C 180,E1 -5298.875,E2 -5298.875} C_VEL
LIN {X 0,Y 509.952,Z 93.278,A -85,B 0,C 180,E1 -5302.079,E2 -5302.079} C_VEL
LIN {X 0,Y 509.981,Z 93.271,A -85,B 0,C 180,E1 -5304.465,E2 -5304.465} C_VEL
LIN {X 0,Y 510.056,Z 93.26,A -85,B 0,C 180,E1 -5307.631,E2 -5307.631} C_VEL
LIN {X 0,Y 510.064,Z 93.257,A -85,B 0,C 180,E1 -5310.79,E2 -5310.79} C_VEL
LIN {X 0,Y 509.954,Z 93.27,A -85,B 0,C 180,E1 -5313.161,E2 -5313.161} C_VEL
LIN {X 0,Y 509.979,Z 93.271,A -85,B 0,C 180,E1 -5316.33,E2 -5316.33} C_VEL
LIN {X 0,Y 509.916,Z 93.275,A -85,B 0,C 180,E1 -5318.721,E2 -5318.721} C_VEL
LIN {X 0,Y 509.906,Z 93.284,A -85,B 0,C 180,E1 -5321.932,E2 -5321.932} C_VEL
LIN {X 0,Y 509.896,Z 93.279,A -85,B 0,C 180,E1 -5325.242,E2 -5325.242} C_VEL
LIN {X 0,Y 509.891,Z 93.283,A -85,B 0,C 180,E1 -5328.001,E2 -5328.001} C_VEL
LIN {X 0,Y 509.853,Z 93.284,A -85,B 0,C 180,E1 -5331.002,E2 -5331.002} C_VEL
LIN {X 0,Y 509.825,Z 93.294,A -85,B 0,C 180,E1 -5333.564,E2 -5333.564} C_VEL
LIN {X 0,Y 509.914,Z 93.276,A -85,B 0,C 180,E1 -5336.379,E2 -5336.379} C_VEL
LIN {X 0,Y 509.879,Z 93.28,A -85,B 0,C 180,E1 -5338.845,E2 -5338.845} C_VEL
LIN {X 0,Y 509.825,Z 93.294,A -85,B 0,C 180,E1 -5341.59,E2 -5341.59} C_VEL
LIN {X 0,Y 509.85,Z 93.283,A -85,B 0,C 180,E1 -5344.414,E2 -5344.414} C_VEL
LIN {X 0,Y 509.818,Z 93.295,A -85,B 0,C 180,E1 -5347.341,E2 -5347.341} C_VEL
LIN {X 0,Y 509.84,Z 93.284,A -85,B 0,C 180,E1 -5350.383,E2 -5350.383} C_VEL
LIN {X 0,Y 509.826,Z 93.292,A -85,B 0,C 180,E1 -5353.063,E2 -5353.063} C_VEL
LIN {X 0,Y 509.833,Z 93.287,A -85,B 0,C 180,E1 -5355.793,E2 -5355.793} C_VEL
LIN {X 0,Y 509.858,Z 93.283,A -85,B 0,C 180,E1 -5358.575,E2 -5358.575} C_VEL
LIN {X 0,Y 509.854,Z 93.284,A -85,B 0,C 180,E1 -5361.787,E2 -5361.787} C_VEL
LIN {X 0,Y 509.839,Z 93.289,A -85,B 0,C 180,E1 -5364.623,E2 -5364.623} C_VEL
LIN {X 0,Y 509.864,Z 93.287,A -85,B 0,C 180,E1 -5367.481,E2 -5367.481} C_VEL
LIN {X 0,Y 509.862,Z 93.286,A -85,B 0,C 180,E1 -5370.274,E2 -5370.274} C_VEL
LIN {X 0,Y 509.9,Z 93.285,A -85,B 0,C 180,E1 -5373.303,E2 -5373.303} C_VEL
LIN {X 0,Y 509.903,Z 93.314,A -85,B 0,C 180,E1 -5373.353,E2 -5373.353} C_VEL
LIN {X 0,Y 510.944,Z 96.203,A -85,B 0,C 180,E1 -5373.46,E2 -5373.46} C_VEL
LIN {X 0,Y 517.888,Z 110.562,A -85,B 0,C 180,E1 -5374.079,E2 -5374.079} C_VEL
LIN {X 0,Y 516.057,Z 256.517,A -85,B 0,C 180,E1 -5376.344,E2 -5376.344} C_VEL
LIN {X 0,Y 515.666,Z 291.422,A -85,B 0,C 180,E1 -5376.905,E2 -5376.905} C_VEL
LIN {X 0,Y 515.303,Z 308.327,A -85,B 0,C 180,E1 -5377.338,E2 -5377.338} C_VEL
LIN {X 0,Y 514.817,Z 325.25,A -85,B 0,C 180,E1 -5377.95,E2 -5377.95} C_VEL
LIN {X 0,Y 514.289,Z 340.67,A -85,B 0,C 180,E1 -5378.675,E2 -5378.675} C_VEL
LIN {X 0,Y 513.702,Z 354.651,A -85,B 0,C 180,E1 -5379.477,E2 -5379.477} C_VEL
LIN {X 0,Y 513.033,Z 369.372,A -85,B 0,C 180,E1 -5380.494,E2 -5380.494} C_VEL
LIN {X 0,Y 512.36,Z 382.914,A -85,B 0,C 180,E1 -5381.61,E2 -5381.61} C_VEL
LIN {X 0,Y 511.703,Z 395.333,A -85,B 0,C 180,E1 -5382.825,E2 -5382.825} C_VEL
LIN {X 0,Y 511.205,Z 406.019,A -85,B 0,C 180,E1 -5384.04,E2 -5384.04} C_VEL
LIN {X 0,Y 510.7,Z 416.737,A -85,B 0,C 180,E1 -5385.455,E2 -5385.455} C_VEL
LIN {X 0,Y 510.235,Z 427.03,A -85,B 0,C 180,E1 -5387.066,E2 -5387.066} C_VEL
LIN {X 0,Y 509.887,Z 435.586,A -85,B 0,C 180,E1 -5388.673,E2 -5388.673} C_VEL
LIN {X 0,Y 509.614,Z 441.909,A -85,B 0,C 180,E1 -5390.073,E2 -5390.073} C_VEL
LIN {X 0,Y 509.463,Z 447.916,A -85,B 0,C 180,E1 -5391.672,E2 -5391.672} C_VEL
LIN {X 0,Y 509.391,Z 453.058,A -85,B 0,C 180,E1 -5393.403,E2 -5393.403} C_VEL
LIN {X 0,Y 509.216,Z 457.172,A -85,B 0,C 180,E1 -5395.25,E2 -5395.25} C_VEL
LIN {X 0,Y 509.271,Z 459.633,A -85,B 0,C 180,E1 -5396.836,E2 -5396.836} C_VEL
LIN {X 0,Y 509.12,Z 461.105,A -85,B 0,C 180,E1 -5398.418,E2 -5398.418} C_VEL
LIN {X 0,Y 509.104,Z 461.665,A -85,B 0,C 180,E1 -5400,E2 -5400} C_VEL
LIN {X 0,Y 509.122,Z 461.217,A -85,B 0,C 180,E1 -5401.582,E2 -5401.582} C_VEL
LIN {X 0,Y 509.273,Z 459.87,A -85,B 0,C 180,E1 -5403.164,E2 -5403.164} C_VEL
LIN {X 0,Y 509.248,Z 457.506,A -85,B 0,C 180,E1 -5404.75,E2 -5404.75} C_VEL
LIN {X 0,Y 509.391,Z 453.517,A -85,B 0,C 180,E1 -5406.596,E2 -5406.596} C_VEL
LIN {X 0,Y 509.495,Z 448.509,A -85,B 0,C 180,E1 -5408.328,E2 -5408.328} C_VEL
LIN {X 0,Y 509.635,Z 442.61,A -85,B 0,C 180,E1 -5409.926,E2 -5409.926} C_VEL
LIN {X 0,Y 509.949,Z 435.42,A -85,B 0,C 180,E1 -5411.527,E2 -5411.527} C_VEL
LIN {X 0,Y 510.309,Z 426.764,A -85,B 0,C 180,E1 -5413.134,E2 -5413.134} C_VEL
LIN {X 0,Y 510.797,Z 416.351,A -85,B 0,C 180,E1 -5414.746,E2 -5414.746} C_VEL
LIN {X 0,Y 511.322,Z 405.488,A -85,B 0,C 180,E1 -5416.161,E2 -5416.161} C_VEL
LIN {X 0,Y 511.794,Z 394.507,A -85,B 0,C 180,E1 -5417.378,E2 -5417.378} C_VEL
LIN {X 0,Y 512.421,Z 381.633,A -85,B 0,C 180,E1 -5418.598,E2 -5418.598} C_VEL
LIN {X 0,Y 513.051,Z 367.662,A -85,B 0,C 180,E1 -5419.714,E2 -5419.714} C_VEL
LIN {X 0,Y 513.609,Z 353.985,A -85,B 0,C 180,E1 -5420.631,E2 -5420.631} C_VEL
LIN {X 0,Y 514.202,Z 339.154,A -85,B 0,C 180,E1 -5421.444,E2 -5421.444} C_VEL
LIN {X 0,Y 514.648,Z 323.647,A -85,B 0,C 180,E1 -5422.131,E2 -5422.131} C_VEL
LIN {X 0,Y 515.049,Z 306.861,A -85,B 0,C 180,E1 -5422.7,E2 -5422.7} C_VEL
LIN {X 0,Y 515.265,Z 290.97,A -85,B 0,C 180,E1 -5423.087,E2 -5423.087} C_VEL
LIN {X 0,Y 517.014,Z 168.455,A -85,B 0,C 180,E1 -5425.067,E2 -5425.067} C_VEL
LIN {X 0,Y 518.117,Z 110.71,A -85,B 0,C 180,E1 -5426.078,E2 -5426.078} C_VEL
LIN {X 0,Y 512.771,Z 99.728,A -85,B 0,C 180,E1 -5426.628,E2 -5426.628} C_VEL
LIN {X 0,Y 509.956,Z 94.154,A -85,B 0,C 180,E1 -5426.932,E2 -5426.932} C_VEL
LIN {X 0,Y 509.795,Z 93.298,A -85,B 0,C 180,E1 -5426.982,E2 -5426.982} C_VEL
LIN {X 0,Y 509.827,Z 93.292,A -85,B 0,C 180,E1 -5429.753,E2 -5429.753} C_VEL
LIN {X 0,Y 509.867,Z 93.29,A -85,B 0,C 180,E1 -5432.772,E2 -5432.772} C_VEL
LIN {X 0,Y 509.824,Z 93.291,A -85,B 0,C 180,E1 -5435.577,E2 -5435.577} C_VEL
LIN {X 0,Y 509.849,Z 93.292,A -85,B 0,C 180,E1 -5438.338,E2 -5438.338} C_VEL
LIN {X 0,Y 509.857,Z 93.286,A -85,B 0,C 180,E1 -5441.425,E2 -5441.425} C_VEL
LIN {X 0,Y 509.84,Z 93.29,A -85,B 0,C 180,E1 -5444.67,E2 -5444.67} C_VEL
LIN {X 0,Y 509.835,Z 93.291,A -85,B 0,C 180,E1 -5447.51,E2 -5447.51} C_VEL
LIN {X 0,Y 509.847,Z 93.289,A -85,B 0,C 180,E1 -5450.647,E2 -5450.647} C_VEL
LIN {X 0,Y 509.826,Z 93.296,A -85,B 0,C 180,E1 -5453.646,E2 -5453.646} C_VEL
LIN {X 0,Y 509.861,Z 93.294,A -85,B 0,C 180,E1 -5456.539,E2 -5456.539} C_VEL
LIN {X 0,Y 509.892,Z 93.341,A -85,B 0,C 180,E1 -5457.522,E2 -5457.522} C_VEL
LIN {X 0,Y 514.633,Z 108.321,A -85,B 0,C 180,E1 -5459.355,E2 -5459.355} C_VEL
LIN {X 0,Y 515.986,Z 113.774,A -85,B 0,C 180,E1 -5459.963,E2 -5459.963} C_VEL
LIN {X 0,Y 514.572,Z 146.706,A -85,B 0,C 180,E1 -5462.91,E2 -5462.91} C_VEL
LIN {X 0,Y 514.472,Z 151.002,A -85,B 0,C 180,E1 -5463.267,E2 -5463.267} C_VEL
LIN {X 0,Y 517.685,Z 174.072,A -85,B 0,C 180,E1 -5463.887,E2 -5463.887} C_VEL
LIN {X 0,Y 515.898,Z 280.064,A -85,B 0,C 180,E1 -5465.637,E2 -5465.637} C_VEL
LIN {X 0,Y 514.992,Z 362.351,A -85,B 0,C 180,E1 -5466.926,E2 -5466.926} C_VEL
LIN {X 0,Y 514.588,Z 379.803,A -85,B 0,C 180,E1 -5467.358,E2 -5467.358} C_VEL
LIN {X 0,Y 514.088,Z 395.995,A -85,B 0,C 180,E1 -5467.917,E2 -5467.917} C_VEL
LIN {X 0,Y 513.551,Z 410.746,A -85,B 0,C 180,E1 -5468.563,E2 -5468.563} C_VEL
LIN {X 0,Y 512.958,Z 425.357,A -85,B 0,C 180,E1 -5469.341,E2 -5469.341} C_VEL
LIN {X 0,Y 512.327,Z 441.058,A -85,B 0,C 180,E1 -5470.361,E2 -5470.361} C_VEL
LIN {X 0,Y 511.678,Z 455.513,A -85,B 0,C 180,E1 -5471.492,E2 -5471.492} C_VEL
LIN {X 0,Y 511.175,Z 468.581,A -85,B 0,C 180,E1 -5472.703,E2 -5472.703} C_VEL
LIN {X 0,Y 510.674,Z 480.771,A -85,B 0,C 180,E1 -5474.023,E2 -5474.023} C_VEL
LIN {X 0,Y 510.321,Z 490.525,A -85,B 0,C 180,E1 -5475.239,E2 -5475.239} C_VEL
LIN {X 0,Y 509.915,Z 501.52,A -85,B 0,C 180,E1 -5476.855,E2 -5476.855} C_VEL
LIN {X 0,Y 509.722,Z 509.404,A -85,B 0,C 180,E1 -5478.22,E2 -5478.22} C_VEL
LIN {X 0,Y 509.498,Z 516.607,A -85,B 0,C 180,E1 -5479.669,E2 -5479.669} C_VEL
LIN {X 0,Y 509.355,Z 523.156,A -85,B 0,C 180,E1 -5481.27,E2 -5481.27} C_VEL
LIN {X 0,Y 509.302,Z 528.537,A -85,B 0,C 180,E1 -5482.865,E2 -5482.865} C_VEL
LIN {X 0,Y 509.26,Z 532.666,A -85,B 0,C 180,E1 -5484.456,E2 -5484.456} C_VEL
LIN {X 0,Y 509.233,Z 535.752,A -85,B 0,C 180,E1 -5486.043,E2 -5486.043} C_VEL
LIN {X 0,Y 509.185,Z 537.762,A -85,B 0,C 180,E1 -5487.626,E2 -5487.626} C_VEL
LIN {X 0,Y 509.087,Z 538.773,A -85,B 0,C 180,E1 -5489.208,E2 -5489.208} C_VEL
LIN {X 0,Y 509.086,Z 538.787,A -85,B 0,C 180,E1 -5490.79,E2 -5490.79} C_VEL
LIN {X 0,Y 509.184,Z 537.819,A -85,B 0,C 180,E1 -5492.373,E2 -5492.373} C_VEL
LIN {X 0,Y 509.233,Z 535.843,A -85,B 0,C 180,E1 -5493.956,E2 -5493.956} C_VEL
LIN {X 0,Y 509.257,Z 532.821,A -85,B 0,C 180,E1 -5495.543,E2 -5495.543} C_VEL
LIN {X 0,Y 509.298,Z 528.746,A -85,B 0,C 180,E1 -5497.134,E2 -5497.134} C_VEL
LIN {X 0,Y 509.354,Z 523.469,A -85,B 0,C 180,E1 -5498.729,E2 -5498.729} C_VEL
LIN {X 0,Y 509.5,Z 517.014,A -85,B 0,C 180,E1 -5500.33,E2 -5500.33} C_VEL
LIN {X 0,Y 509.754,Z 509.151,A -85,B 0,C 180,E1 -5501.935,E2 -5501.935} C_VEL
LIN {X 0,Y 510.045,Z 499.703,A -85,B 0,C 180,E1 -5503.547,E2 -5503.547} C_VEL
LIN {X 0,Y 510.409,Z 489.967,A -85,B 0,C 180,E1 -5504.961,E2 -5504.961} C_VEL
LIN {X 0,Y 510.909,Z 478.598,A -85,B 0,C 180,E1 -5506.379,E2 -5506.379} C_VEL
LIN {X 0,Y 511.541,Z 465.14,A -85,B 0,C 180,E1 -5507.799,E2 -5507.799} C_VEL
LIN {X 0,Y 512.168,Z 451.098,A -85,B 0,C 180,E1 -5509.047,E2 -5509.047} C_VEL
LIN {X 0,Y 512.864,Z 436.415,A -85,B 0,C 180,E1 -5510.138,E2 -5510.138} C_VEL
LIN {X 0,Y 513.499,Z 422.286,A -85,B 0,C 180,E1 -5511.018,E2 -5511.018} C_VEL
LIN {X 0,Y 514.12,Z 406.763,A -85,B 0,C 180,E1 -5511.817,E2 -5511.817} C_VEL
LIN {X 0,Y 514.767,Z 390.664,A -85,B 0,C 180,E1 -5512.474,E2 -5512.474} C_VEL
LIN {X 0,Y 515.252,Z 374.079,A -85,B 0,C 180,E1 -5512.981,E2 -5512.981} C_VEL
LIN {X 0,Y 515.635,Z 357.23,A -85,B 0,C 180,E1 -5513.33,E2 -5513.33} C_VEL
LIN {X 0,Y 517.862,Z 174.311,A -85,B 0,C 180,E1 -5516.146,E2 -5516.146} C_VEL
LIN {X 0,Y 515.018,Z 154.987,A -85,B 0,C 180,E1 -5516.639,E2 -5516.639} C_VEL
LIN {X 0,Y 516.272,Z 121.538,A -85,B 0,C 180,E1 -5519.568,E2 -5519.568} C_VEL
LIN {X 0,Y 516.422,Z 114.111,A -85,B 0,C 180,E1 -5520.233,E2 -5520.233} C_VEL
LIN {X 0,Y 509.864,Z 93.291,A -85,B 0,C 180,E1 -5522.586,E2 -5522.586} C_VEL
LIN {X 0,Y 509.824,Z 93.29,A -85,B 0,C 180,E1 -5525.578,E2 -5525.578} C_VEL
LIN {X 0,Y 509.845,Z 93.292,A -85,B 0,C 180,E1 -5528.338,E2 -5528.338} C_VEL
LIN {X 0,Y 509.853,Z 93.285,A -85,B 0,C 180,E1 -5531.425,E2 -5531.425} C_VEL
LIN {X 0,Y 509.852,Z 93.29,A -85,B 0,C 180,E1 -5534.668,E2 -5534.668} C_VEL
LIN {X 0,Y 509.852,Z 93.288,A -85,B 0,C 180,E1 -5538.103,E2 -5538.103} C_VEL
LIN {X 0,Y 509.843,Z 93.288,A -85,B 0,C 180,E1 -5540.648,E2 -5540.648} C_VEL
LIN {X 0,Y 509.831,Z 93.287,A -85,B 0,C 180,E1 -5543.648,E2 -5543.648} C_VEL
LIN {X 0,Y 509.857,Z 93.287,A -85,B 0,C 180,E1 -5546.539,E2 -5546.539} C_VEL
LIN {X 0,Y 509.845,Z 93.284,A -85,B 0,C 180,E1 -5549.334,E2 -5549.334} C_VEL
LIN {X 0,Y 509.889,Z 93.287,A -85,B 0,C 180,E1 -5552.054,E2 -5552.054} C_VEL
LIN {X 0,Y 509.873,Z 93.282,A -85,B 0,C 180,E1 -5554.704,E2 -5554.704} C_VEL
LIN {X 0,Y 509.832,Z 93.287,A -85,B 0,C 180,E1 -5557.455,E2 -5557.455} C_VEL
LIN {X 0,Y 509.912,Z 93.282,A -85,B 0,C 180,E1 -5559.845,E2 -5559.845} C_VEL
LIN {X 0,Y 509.88,Z 93.28,A -85,B 0,C 180,E1 -5563.175,E2 -5563.175} C_VEL
LIN {X 0,Y 509.86,Z 93.287,A -85,B 0,C 180,E1 -5565.634,E2 -5565.634} C_VEL
LIN {X 0,Y 509.918,Z 93.275,A -85,B 0,C 180,E1 -5568.875,E2 -5568.875} C_VEL
LIN {X 0,Y 509.947,Z 93.276,A -85,B 0,C 180,E1 -5572.078,E2 -5572.078} C_VEL
LIN {X 0,Y 509.977,Z 93.268,A -85,B 0,C 180,E1 -5574.464,E2 -5574.464} C_VEL
LIN {X 0,Y 510.05,Z 93.267,A -85,B 0,C 180,E1 -5577.631,E2 -5577.631} C_VEL
LIN {X 0,Y 510.06,Z 93.257,A -85,B 0,C 180,E1 -5580.79,E2 -5580.79} C_VEL
LIN {X 0,Y 509.952,Z 93.274,A -85,B 0,C 180,E1 -5583.16,E2 -5583.16} C_VEL
LIN {X 0,Y 509.974,Z 93.268,A -85,B 0,C 180,E1 -5586.33,E2 -5586.33} C_VEL
LIN {X 0,Y 509.91,Z 93.276,A -85,B 0,C 180,E1 -5588.72,E2 -5588.72} C_VEL
LIN {X 0,Y 509.9,Z 93.279,A -85,B 0,C 180,E1 -5591.932,E2 -5591.932} C_VEL
LIN {X 0,Y 509.889,Z 93.286,A -85,B 0,C 180,E1 -5595.242,E2 -5595.242} C_VEL
LIN {X 0,Y 509.885,Z 93.28,A -85,B 0,C 180,E1 -5598.001,E2 -5598.001} C_VEL
LIN {X 0,Y 509.846,Z 93.289,A -85,B 0,C 180,E1 -5601.002,E2 -5601.002} C_VEL
LIN {X 0,Y 509.833,Z 93.289,A -85,B 0,C 180,E1 -5603.563,E2 -5603.563} C_VEL
LIN {X 0,Y 509.908,Z 93.276,A -85,B 0,C 180,E1 -5606.379,E2 -5606.379} C_VEL
LIN {X 0,Y 509.873,Z 93.285,A -85,B 0,C 180,E1 -5608.844,E2 -5608.844} C_VEL
LIN {X 0,Y 509.821,Z 93.289,A -85,B 0,C 180,E1 -5611.59,E2 -5611.59} C_VEL
LIN {X 0,Y 509.85,Z 93.285,A -85,B 0,C 180,E1 -5614.414,E2 -5614.414} C_VEL
LIN {X 0,Y 509.816,Z 93.291,A -85,B 0,C 180,E1 -5617.341,E2 -5617.341} C_VEL
LIN {X 0,Y 509.835,Z 93.287,A -85,B 0,C 180,E1 -5620.382,E2 -5620.382} C_VEL
LIN {X 0,Y 509.835,Z 93.291,A -85,B 0,C 180,E1 -5623.065,E2 -5623.065} C_VEL
LIN {X 0,Y 509.827,Z 93.286,A -85,B 0,C 180,E1 -5625.793,E2 -5625.793} C_VEL
LIN {X 0,Y 509.856,Z 93.288,A -85,B 0,C 180,E1 -5628.575,E2 -5628.575} C_VEL
LIN {X 0,Y 509.848,Z 93.283,A -85,B 0,C 180,E1 -5631.787,E2 -5631.787} C_VEL
LIN {X 0,Y 509.817,Z 93.287,A -85,B 0,C 180,E1 -5633.738,E2 -5633.738} C_VEL
LIN {X 0,Y 509.149,Z 93.377,A -85,B 0,C 180,E1 -5634.397,E2 -5634.397} C_VEL
LIN {X 0,Y 506.337,Z 93.726,A -85,B 0,C 180,E1 -5635.469,E2 -5635.469} C_VEL
LIN {X 0,Y 503.95,Z 94.024,A -85,B 0,C 180,E1 -5636.333,E2 -5636.333} C_VEL
LIN {X 0,Y 502.904,Z 94.153,A -85,B 0,C 180,E1 -5636.999,E2 -5636.999} C_VEL
LIN {X 0,Y 502.806,Z 94.162,A -85,B 0,C 180,E1 -5637.225,E2 -5637.225} C_VEL
LIN {X 0,Y 502.813,Z 94.162,A -85,B 0,C 180,E1 -5640.065,E2 -5640.065} C_VEL
LIN {X 0,Y 502.832,Z 94.167,A -85,B 0,C 180,E1 -5642.534,E2 -5642.534} C_VEL
LIN {X 0,Y 502.828,Z 94.158,A -85,B 0,C 180,E1 -5645.299,E2 -5645.299} C_VEL
LIN {X 0,Y 502.78,Z 94.165,A -85,B 0,C 180,E1 -5647.827,E2 -5647.827} C_VEL
LIN {X 0,Y 502.825,Z 94.168,A -85,B 0,C 180,E1 -5650.401,E2 -5650.401} C_VEL
LIN {X 0,Y 502.833,Z 94.159,A -85,B 0,C 180,E1 -5652.932,E2 -5652.932} C_VEL
LIN {X 0,Y 502.845,Z 94.156,A -85,B 0,C 180,E1 -5655.43,E2 -5655.43} C_VEL
LIN {X 0,Y 502.877,Z 94.155,A -85,B 0,C 180,E1 -5658.717,E2 -5658.717} C_VEL
LIN {X 0,Y 502.902,Z 94.154,A -85,B 0,C 180,E1 -5661.967,E2 -5661.967} C_VEL
LIN {X 0,Y 502.938,Z 94.15,A -85,B 0,C 180,E1 -5664.387,E2 -5664.387} C_VEL
LIN {X 0,Y 503.025,Z 94.136,A -85,B 0,C 180,E1 -5667.598,E2 -5667.598} C_VEL
LIN {X 0,Y 503.028,Z 94.141,A -85,B 0,C 180,E1 -5670.001,E2 -5670.001} C_VEL
LIN {X 0,Y 503.026,Z 94.137,A -85,B 0,C 180,E1 -5672.403,E2 -5672.403} C_VEL
LIN {X 0,Y 502.938,Z 94.148,A -85,B 0,C 180,E1 -5675.614,E2 -5675.614} C_VEL
LIN {X 0,Y 502.903,Z 94.156,A -85,B 0,C 180,E1 -5678.034,E2 -5678.034} C_VEL
LIN {X 0,Y 502.879,Z 94.153,A -85,B 0,C 180,E1 -5681.284,E2 -5681.284} C_VEL
LIN {X 0,Y 502.847,Z 94.156,A -85,B 0,C 180,E1 -5684.571,E2 -5684.571} C_VEL
LIN {X 0,Y 502.864,Z 94.16,A -85,B 0,C 180,E1 -5687.907,E2 -5687.907} C_VEL
LIN {X 0,Y 502.831,Z 94.158,A -85,B 0,C 180,E1 -5690.537,E2 -5690.537} C_VEL
LIN {X 0,Y 502.79,Z 94.164,A -85,B 0,C 180,E1 -5693.041,E2 -5693.041} C_VEL
LIN {X 0,Y 502.824,Z 94.167,A -85,B 0,C 180,E1 -5695.677,E2 -5695.677} C_VEL
LIN {X 0,Y 502.843,Z 94.157,A -85,B 0,C 180,E1 -5698.373,E2 -5698.373} C_VEL
LIN {X 0,Y 502.797,Z 94.171,A -85,B 0,C 180,E1 -5701.499,E2 -5701.499} C_VEL
LIN {X 0,Y 502.806,Z 94.163,A -85,B 0,C 180,E1 -5703.994,E2 -5703.994} C_VEL
LIN {X 0,Y 502.779,Z 94.169,A -85,B 0,C 180,E1 -5707.178,E2 -5707.178} C_VEL
LIN {X 0,Y 502.79,Z 94.164,A -85,B 0,C 180,E1 -5710.016,E2 -5710.016} C_VEL
LIN {X 0,Y 502.806,Z 94.161,A -85,B 0,C 180,E1 -5712.2,E2 -5712.2} C_VEL
LIN {X 0,Y 502.804,Z 94.167,A -85,B 0,C 180,E1 -5715.469,E2 -5715.469} C_VEL
LIN {X 0,Y 502.822,Z 94.164,A -85,B 0,C 180,E1 -5718.934,E2 -5718.934} C_VEL
LIN {X 0,Y 502.796,Z 94.162,A -85,B 0,C 180,E1 -5722.046,E2 -5722.046} C_VEL
LIN {X 0,Y 502.807,Z 94.168,A -85,B 0,C 180,E1 -5725.035,E2 -5725.035} C_VEL
LIN {X 0,Y 502.787,Z 94.166,A -85,B 0,C 180,E1 -5727.916,E2 -5727.916} C_VEL
LIN {X 0,Y 502.828,Z 94.166,A -85,B 0,C 180,E1 -5730.712,E2 -5730.712} C_VEL
LIN {X 0,Y 502.882,Z 94.35,A -85,B 0,C 180,E1 -5732.97,E2 -5732.97} C_VEL
LIN {X 0,Y 504.056,Z 97.337,A -85,B 0,C 180,E1 -5733.09,E2 -5733.09} C_VEL
LIN {X 0,Y 511.446,Z 112.578,A -85,B 0,C 180,E1 -5733.765,E2 -5733.765} C_VEL
LIN {X 0,Y 509.512,Z 255.988,A -85,B 0,C 180,E1 -5736.038,E2 -5736.038} C_VEL
LIN {X 0,Y 509.072,Z 291.539,A -85,B 0,C 180,E1 -5736.615,E2 -5736.615} C_VEL
LIN {X 0,Y 508.692,Z 308.472,A -85,B 0,C 180,E1 -5737.054,E2 -5737.054} C_VEL
LIN {X 0,Y 508.149,Z 325.821,A -85,B 0,C 180,E1 -5737.688,E2 -5737.688} C_VEL
LIN {X 0,Y 507.603,Z 341.068,A -85,B 0,C 180,E1 -5738.415,E2 -5738.415} C_VEL
LIN {X 0,Y 506.91,Z 356.122,A -85,B 0,C 180,E1 -5739.296,E2 -5739.296} C_VEL
LIN {X 0,Y 506.215,Z 370.658,A -85,B 0,C 180,E1 -5740.326,E2 -5740.326} C_VEL
LIN {X 0,Y 505.502,Z 384.093,A -85,B 0,C 180,E1 -5741.456,E2 -5741.456} C_VEL
LIN {X 0,Y 504.766,Z 397.418,A -85,B 0,C 180,E1 -5742.79,E2 -5742.79} C_VEL
LIN {X 0,Y 504.159,Z 408.69,A -85,B 0,C 180,E1 -5744.127,E2 -5744.127} C_VEL
LIN {X 0,Y 503.623,Z 419.705,A -85,B 0,C 180,E1 -5745.659,E2 -5745.659} C_VEL
LIN {X 0,Y 503.154,Z 429.603,A -85,B 0,C 180,E1 -5747.291,E2 -5747.291} C_VEL
LIN {X 0,Y 502.851,Z 436.947,A -85,B 0,C 180,E1 -5748.716,E2 -5748.716} C_VEL
LIN {X 0,Y 502.559,Z 443.904,A -85,B 0,C 180,E1 -5750.339,E2 -5750.339} C_VEL
LIN {X 0,Y 502.399,Z 449.627,A -85,B 0,C 180,E1 -5751.959,E2 -5751.959} C_VEL
LIN {X 0,Y 502.325,Z 454.204,A -85,B 0,C 180,E1 -5753.573,E2 -5753.573} C_VEL
LIN {X 0,Y 502.144,Z 457.664,A -85,B 0,C 180,E1 -5755.183,E2 -5755.183} C_VEL
LIN {X 0,Y 502.215,Z 460.154,A -85,B 0,C 180,E1 -5756.791,E2 -5756.791} C_VEL
LIN {X 0,Y 502.044,Z 461.626,A -85,B 0,C 180,E1 -5758.396,E2 -5758.396} C_VEL
LIN {X 0,Y 502.025,Z 462.206,A -85,B 0,C 180,E1 -5760,E2 -5760} C_VEL
LIN {X 0,Y 502.045,Z 461.753,A -85,B 0,C 180,E1 -5761.604,E2 -5761.604} C_VEL
LIN {X 0,Y 502.217,Z 460.42,A -85,B 0,C 180,E1 -5763.209,E2 -5763.209} C_VEL
LIN {X 0,Y 502.193,Z 458.04,A -85,B 0,C 180,E1 -5764.817,E2 -5764.817} C_VEL
LIN {X 0,Y 502.329,Z 454.243,A -85,B 0,C 180,E1 -5766.609,E2 -5766.609} C_VEL
LIN {X 0,Y 502.449,Z 449.002,A -85,B 0,C 180,E1 -5768.445,E2 -5768.445} C_VEL
LIN {X 0,Y 502.625,Z 443.083,A -85,B 0,C 180,E1 -5770.066,E2 -5770.066} C_VEL
LIN {X 0,Y 502.938,Z 436.487,A -85,B 0,C 180,E1 -5771.559,E2 -5771.559} C_VEL
LIN {X 0,Y 503.29,Z 428.356,A -85,B 0,C 180,E1 -5773.115,E2 -5773.115} C_VEL
LIN {X 0,Y 503.808,Z 418.096,A -85,B 0,C 180,E1 -5774.749,E2 -5774.749} C_VEL
LIN {X 0,Y 504.335,Z 407.381,A -85,B 0,C 180,E1 -5776.183,E2 -5776.183} C_VEL
LIN {X 0,Y 504.864,Z 396.644,A -85,B 0,C 180,E1 -5777.415,E2 -5777.415} C_VEL
LIN {X 0,Y 505.497,Z 384.116,A -85,B 0,C 180,E1 -5778.649,E2 -5778.649} C_VEL
LIN {X 0,Y 506.173,Z 370.483,A -85,B 0,C 180,E1 -5779.781,E2 -5779.781} C_VEL
LIN {X 0,Y 506.849,Z 355.504,A -85,B 0,C 180,E1 -5780.813,E2 -5780.813} C_VEL
LIN {X 0,Y 507.425,Z 341.009,A -85,B 0,C 180,E1 -5781.634,E2 -5781.634} C_VEL
LIN {X 0,Y 507.939,Z 325.021,A -85,B 0,C 180,E1 -5782.364,E2 -5782.364} C_VEL
LIN {X 0,Y 508.372,Z 308.76,A -85,B 0,C 180,E1 -5782.934,E2 -5782.934} C_VEL
LIN {X 0,Y 508.635,Z 292.304,A -85,B 0,C 180,E1 -5783.352,E2 -5783.352} C_VEL
LIN {X 0,Y 510.551,Z 173.355,A -85,B 0,C 180,E1 -5785.333,E2 -5785.333} C_VEL
LIN {X 0,Y 511.883,Z 112.817,A -85,B 0,C 180,E1 -5786.42,E2 -5786.42} C_VEL
LIN {X 0,Y 505.968,Z 100.917,A -85,B 0,C 180,E1 -5787.069,E2 -5787.069} C_VEL
LIN {X 0,Y 502.969,Z 95.148,A -85,B 0,C 180,E1 -5787.408,E2 -5787.408} C_VEL
LIN {X 0,Y 502.771,Z 94.173,A -85,B 0,C 180,E1 -5787.47,E2 -5787.47} C_VEL
LIN {X 0,Y 502.789,Z 94.17,A -85,B 0,C 180,E1 -5790.212,E2 -5790.212} C_VEL
LIN {X 0,Y 502.831,Z 94.166,A -85,B 0,C 180,E1 -5793.031,E2 -5793.031} C_VEL
LIN {X 0,Y 502.769,Z 94.172,A -85,B 0,C 180,E1 -5795.951,E2 -5795.951} C_VEL
LIN {X 0,Y 502.795,Z 94.168,A -85,B 0,C 180,E1 -5798.976,E2 -5798.976} C_VEL
LIN {X 0,Y 502.821,Z 94.163,A -85,B 0,C 180,E1 -5801.066,E2 -5801.066} C_VEL
LIN {X 0,Y 502.787,Z 94.17,A -85,B 0,C 180,E1 -5804.53,E2 -5804.53} C_VEL
LIN {X 0,Y 502.797,Z 94.17,A -85,B 0,C 180,E1 -5807.86,E2 -5807.86} C_VEL
LIN {X 0,Y 502.803,Z 94.166,A -85,B 0,C 180,E1 -5811.023,E2 -5811.023} C_VEL
LIN {X 0,Y 502.776,Z 94.174,A -85,B 0,C 180,E1 -5814.169,E2 -5814.169} C_VEL
LIN {X 0,Y 502.829,Z 94.23,A -85,B 0,C 180,E1 -5817.041,E2 -5817.041} C_VEL
LIN {X 0,Y 507.112,Z 107.094,A -85,B 0,C 180,E1 -5818.712,E2 -5818.712} C_VEL
LIN {X 0,Y 509.463,Z 116.122,A -85,B 0,C 180,E1 -5819.767,E2 -5819.767} C_VEL
LIN {X 0,Y 508.029,Z 145.423,A -85,B 0,C 180,E1 -5822.445,E2 -5822.445} C_VEL
LIN {X 0,Y 507.868,Z 149.683,A -85,B 0,C 180,E1 -5822.828,E2 -5822.828} C_VEL
LIN {X 0,Y 510.696,Z 169.625,A -85,B 0,C 180,E1 -5823.399,E2 -5823.399} C_VEL
LIN {X 0,Y 511.369,Z 175.869,A -85,B 0,C 180,E1 -5823.557,E2 -5823.557} C_VEL
LIN {X 0,Y 509.374,Z 278.146,A -85,B 0,C 180,E1 -5825.304,E2 -5825.304} C_VEL
LIN {X 0,Y 508.305,Z 361.987,A -85,B 0,C 180,E1 -5826.658,E2 -5826.658} C_VEL
LIN {X 0,Y 507.891,Z 378.328,A -85,B 0,C 180,E1 -5827.069,E2 -5827.069} C_VEL
LIN {X 0,Y 507.313,Z 395.34,A -85,B 0,C 180,E1 -5827.66,E2 -5827.66} C_VEL
LIN {X 0,Y 506.706,Z 410.851,A -85,B 0,C 180,E1 -5828.353,E2 -5828.353} C_VEL
LIN {X 0,Y 506.007,Z 427.123,A -85,B 0,C 180,E1 -5829.257,E2 -5829.257} C_VEL
LIN {X 0,Y 505.33,Z 442.414,A -85,B 0,C 180,E1 -5830.289,E2 -5830.289} C_VEL
LIN {X 0,Y 504.644,Z 456.524,A -85,B 0,C 180,E1 -5831.423,E2 -5831.423} C_VEL
LIN {X 0,Y 504.077,Z 470.531,A -85,B 0,C 180,E1 -5832.766,E2 -5832.766} C_VEL
LIN {X 0,Y 503.533,Z 482.898,A -85,B 0,C 180,E1 -5834.17,E2 -5834.17} C_VEL
LIN {X 0,Y 503.129,Z 493.929,A -85,B 0,C 180,E1 -5835.644,E2 -5835.644} C_VEL
LIN {X 0,Y 502.768,Z 504.308,A -85,B 0,C 180,E1 -5837.281,E2 -5837.281} C_VEL
LIN {X 0,Y 502.534,Z 512.043,A -85,B 0,C 180,E1 -5838.709,E2 -5838.709} C_VEL
LIN {X 0,Y 502.284,Z 519.32,A -85,B 0,C 180,E1 -5840.333,E2 -5840.333} C_VEL
LIN {X 0,Y 502.245,Z 525.324,A -85,B 0,C 180,E1 -5841.956,E2 -5841.956} C_VEL
LIN {X 0,Y 502.212,Z 530.143,A -85,B 0,C 180,E1 -5843.572,E2 -5843.572} C_VEL
LIN {X 0,Y 502.073,Z 533.726,A -85,B 0,C 180,E1 -5845.182,E2 -5845.182} C_VEL
LIN {X 0,Y 502.141,Z 536.36,A -85,B 0,C 180,E1 -5846.79,E2 -5846.79} C_VEL
LIN {X 0,Y 502.036,Z 537.826,A -85,B 0,C 180,E1 -5848.395,E2 -5848.395} C_VEL
LIN {X 0,Y 502.002,Z 538.407,A -85,B 0,C 180,E1 -5849.999,E2 -5849.999} C_VEL
LIN {X 0,Y 502.034,Z 537.882,A -85,B 0,C 180,E1 -5851.604,E2 -5851.604} C_VEL
LIN {X 0,Y 502.115,Z 536.46,A -85,B 0,C 180,E1 -5853.209,E2 -5853.209} C_VEL
LIN {X 0,Y 502.067,Z 533.909,A -85,B 0,C 180,E1 -5854.817,E2 -5854.817} C_VEL
LIN {X 0,Y 502.186,Z 530.268,A -85,B 0,C 180,E1 -5856.472,E2 -5856.472} C_VEL
LIN {X 0,Y 502.245,Z 525.683,A -85,B 0,C 180,E1 -5858.043,E2 -5858.043} C_VEL
LIN {X 0,Y 502.283,Z 519.802,A -85,B 0,C 180,E1 -5859.665,E2 -5859.665} C_VEL
LIN {X 0,Y 502.54,Z 512.669,A -85,B 0,C 180,E1 -5861.29,E2 -5861.29} C_VEL
LIN {X 0,Y 502.802,Z 503.982,A -85,B 0,C 180,E1 -5862.922,E2 -5862.922} C_VEL
LIN {X 0,Y 503.237,Z 493.632,A -85,B 0,C 180,E1 -5864.559,E2 -5864.559} C_VEL
LIN {X 0,Y 503.734,Z 482.859,A -85,B 0,C 180,E1 -5866.004,E2 -5866.004} C_VEL
LIN {X 0,Y 504.287,Z 470.369,A -85,B 0,C 180,E1 -5867.435,E2 -5867.435} C_VEL
LIN {X 0,Y 504.958,Z 456.939,A -85,B 0,C 180,E1 -5868.74,E2 -5868.74} C_VEL
LIN {X 0,Y 505.694,Z 442.689,A -85,B 0,C 180,E1 -5869.906,E2 -5869.906} C_VEL
LIN {X 0,Y 506.409,Z 427.57,A -85,B 0,C 180,E1 -5870.938,E2 -5870.938} C_VEL
LIN {X 0,Y 507.169,Z 412.023,A -85,B 0,C 180,E1 -5871.808,E2 -5871.808} C_VEL
LIN {X 0,Y 507.84,Z 395.997,A -85,B 0,C 180,E1 -5872.529,E2 -5872.529} C_VEL
LIN {X 0,Y 508.428,Z 379.768,A -85,B 0,C 180,E1 -5873.093,E2 -5873.093} C_VEL
LIN {X 0,Y 508.896,Z 363.514,A -85,B 0,C 180,E1 -5873.501,E2 -5873.501} C_VEL
LIN {X 0,Y 511.444,Z 174.805,A -85,B 0,C 180,E1 -5876.484,E2 -5876.484} C_VEL
LIN {X 0,Y 508.399,Z 154.676,A -85,B 0,C 180,E1 -5877.005,E2 -5877.005} C_VEL
LIN {X 0,Y 509.87,Z 119.861,A -85,B 0,C 180,E1 -5880.091,E2 -5880.091} C_VEL
LIN {X 0,Y 509.798,Z 116.14,A -85,B 0,C 180,E1 -5880.439,E2 -5880.439} C_VEL
LIN {X 0,Y 502.818,Z 94.167,A -85,B 0,C 180,E1 -5882.959,E2 -5882.959} C_VEL
LIN {X 0,Y 502.77,Z 94.17,A -85,B 0,C 180,E1 -5885.951,E2 -5885.951} C_VEL
LIN {X 0,Y 502.797,Z 94.168,A -85,B 0,C 180,E1 -5888.976,E2 -5888.976} C_VEL
LIN {X 0,Y 502.826,Z 94.166,A -85,B 0,C 180,E1 -5892.202,E2 -5892.202} C_VEL
LIN {X 0,Y 502.796,Z 94.164,A -85,B 0,C 180,E1 -5895.468,E2 -5895.468} C_VEL
LIN {X 0,Y 502.815,Z 94.161,A -85,B 0,C 180,E1 -5898.934,E2 -5898.934} C_VEL
LIN {X 0,Y 502.79,Z 94.168,A -85,B 0,C 180,E1 -5902.046,E2 -5902.046} C_VEL
LIN {X 0,Y 502.805,Z 94.161,A -85,B 0,C 180,E1 -5905.035,E2 -5905.035} C_VEL
LIN {X 0,Y 502.781,Z 94.169,A -85,B 0,C 180,E1 -5907.915,E2 -5907.915} C_VEL
LIN {X 0,Y 502.822,Z 94.161,A -85,B 0,C 180,E1 -5910.712,E2 -5910.712} C_VEL
LIN {X 0,Y 502.858,Z 94.155,A -85,B 0,C 180,E1 -5913.439,E2 -5913.439} C_VEL
LIN {X 0,Y 502.788,Z 94.172,A -85,B 0,C 180,E1 -5916.086,E2 -5916.086} C_VEL
LIN {X 0,Y 502.779,Z 94.165,A -85,B 0,C 180,E1 -5918.689,E2 -5918.689} C_VEL
LIN {X 0,Y 502.826,Z 94.159,A -85,B 0,C 180,E1 -5921.248,E2 -5921.248} C_VEL
LIN {X 0,Y 502.818,Z 94.166,A -85,B 0,C 180,E1 -5923.767,E2 -5923.767} C_VEL
LIN {X 0,Y 502.827,Z 94.162,A -85,B 0,C 180,E1 -5926.255,E2 -5926.255} C_VEL
LIN {X 0,Y 502.888,Z 94.151,A -85,B 0,C 180,E1 -5928.717,E2 -5928.717} C_VEL
LIN {X 0,Y 502.897,Z 94.155,A -85,B 0,C 180,E1 -5931.967,E2 -5931.967} C_VEL
LIN {X 0,Y 502.933,Z 94.146,A -85,B 0,C 180,E1 -5934.387,E2 -5934.387} C_VEL
LIN {X 0,Y 503.02,Z 94.142,A -85,B 0,C 180,E1 -5937.598,E2 -5937.598} C_VEL
LIN {X 0,Y 503.023,Z 94.137,A -85,B 0,C 180,E1 -5940,E2 -5940} C_VEL
LIN {X 0,Y 503.021,Z 94.134,A -85,B 0,C 180,E1 -5942.402,E2 -5942.402} C_VEL
LIN {X 0,Y 502.933,Z 94.153,A -85,B 0,C 180,E1 -5945.614,E2 -5945.614} C_VEL
LIN {X 0,Y 502.897,Z 94.151,A -85,B 0,C 180,E1 -5948.033,E2 -5948.033} C_VEL
LIN {X 0,Y 502.873,Z 94.159,A -85,B 0,C 180,E1 -5951.283,E2 -5951.283} C_VEL
LIN {X 0,Y 502.841,Z 94.157,A -85,B 0,C 180,E1 -5954.571,E2 -5954.571} C_VEL
LIN {X 0,Y 502.858,Z 94.156,A -85,B 0,C 180,E1 -5957.907,E2 -5957.907} C_VEL
LIN {X 0,Y 502.824,Z 94.159,A -85,B 0,C 180,E1 -5960.536,E2 -5960.536} C_VEL
LIN {X 0,Y 502.793,Z 94.168,A -85,B 0,C 180,E1 -5963.041,E2 -5963.041} C_VEL
LIN {X 0,Y 502.836,Z 94.159,A -85,B 0,C 180,E1 -5965.676,E2 -5965.676} C_VEL
LIN {X 0,Y 502.836,Z 94.158,A -85,B 0,C 180,E1 -5968.373,E2 -5968.373} C_VEL
LIN {X 0,Y 502.792,Z 94.166,A -85,B 0,C 180,E1 -5971.5,E2 -5971.5} C_VEL
LIN {X 0,Y 502.803,Z 94.163,A -85,B 0,C 180,E1 -5974.445,E2 -5974.445} C_VEL
LIN {X 0,Y 502.778,Z 94.17,A -85,B 0,C 180,E1 -5977.179,E2 -5977.179} C_VEL
LIN {X 0,Y 502.785,Z 94.163,A -85,B 0,C 180,E1 -5980.015,E2 -5980.015} C_VEL
LIN {X 0,Y 502.799,Z 94.162,A -85,B 0,C 180,E1 -5982.2,E2 -5982.2} C_VEL
LIN {X 0,Y 502.797,Z 94.163,A -85,B 0,C 180,E1 -5985.469,E2 -5985.469} C_VEL
LIN {X 0,Y 502.827,Z 94.158,A -85,B 0,C 180,E1 -5987.865,E2 -5987.865} C_VEL
LIN {X 0,Y 502.8,Z 94.166,A -85,B 0,C 180,E1 -5991.025,E2 -5991.025} C_VEL
LIN {X 0,Y 502.772,Z 94.167,A -85,B 0,C 180,E1 -5994.17,E2 -5994.17} C_VEL
LIN {X 0,Y 502.806,Z 94.162,A -85,B 0,C 180,E1 -5997.225,E2 -5997.225} C_VEL
LIN {X 0,Y 502.105,Z 94.249,A -85,B 0,C 180,E1 -5997.894,E2 -5997.894} C_VEL
LIN {X 0,Y 499.24,Z 94.608,A -85,B 0,C 180,E1 -5998.979,E2 -5998.979} C_VEL
LIN {X 0,Y 496.846,Z 94.906,A -85,B 0,C 180,E1 -5999.854,E2 -5999.854} C_VEL
LIN {X 0,Y 495.829,Z 95.038,A -85,B 0,C 180,E1 -6000.53,E2 -6000.53} C_VEL
LIN {X 0,Y 495.751,Z 95.04,A -85,B 0,C 180,E1 -6000.759,E2 -6000.759} C_VEL
LIN {X 0,Y 495.789,Z 95.036,A -85,B 0,C 180,E1 -6003.933,E2 -6003.933} C_VEL
LIN {X 0,Y 495.76,Z 95.039,A -85,B 0,C 180,E1 -6007.139,E2 -6007.139} C_VEL
LIN {X 0,Y 495.771,Z 95.042,A -85,B 0,C 180,E1 -6010.11,E2 -6010.11} C_VEL
LIN {X 0,Y 495.786,Z 95.039,A -85,B 0,C 180,E1 -6012.682,E2 -6012.682} C_VEL
LIN {X 0,Y 495.79,Z 95.035,A -85,B 0,C 180,E1 -6015.218,E2 -6015.218} C_VEL
LIN {X 0,Y 495.852,Z 95.032,A -85,B 0,C 180,E1 -6018.555,E2 -6018.555} C_VEL
LIN {X 0,Y 495.873,Z 95.028,A -85,B 0,C 180,E1 -6021.853,E2 -6021.853} C_VEL
LIN {X 0,Y 495.895,Z 95.028,A -85,B 0,C 180,E1 -6024.307,E2 -6024.307} C_VEL
LIN {X 0,Y 495.994,Z 95.011,A -85,B 0,C 180,E1 -6027.564,E2 -6027.564} C_VEL
LIN {X 0,Y 495.984,Z 95.011,A -85,B 0,C 180,E1 -6030.812,E2 -6030.812} C_VEL
LIN {X 0,Y 495.994,Z 95.012,A -85,B 0,C 180,E1 -6032.437,E2 -6032.437} C_VEL
LIN {X 0,Y 495.896,Z 95.026,A -85,B 0,C 180,E1 -6035.694,E2 -6035.694} C_VEL
LIN {X 0,Y 495.874,Z 95.03,A -85,B 0,C 180,E1 -6038.148,E2 -6038.148} C_VEL
LIN {X 0,Y 495.853,Z 95.03,A -85,B 0,C 180,E1 -6041.446,E2 -6041.446} C_VEL
LIN {X 0,Y 495.792,Z 95.035,A -85,B 0,C 180,E1 -6044.783,E2 -6044.783} C_VEL
LIN {X 0,Y 495.788,Z 95.038,A -85,B 0,C 180,E1 -6047.319,E2 -6047.319} C_VEL
LIN {X 0,Y 495.774,Z 95.043,A -85,B 0,C 180,E1 -6049.891,E2 -6049.891} C_VEL
LIN {X 0,Y 495.761,Z 95.039,A -85,B 0,C 180,E1 -6052.861,E2 -6052.861} C_VEL
LIN {X 0,Y 495.783,Z 95.038,A -85,B 0,C 180,E1 -6056.069,E2 -6056.069} C_VEL
LIN {X 0,Y 495.774,Z 95.037,A -85,B 0,C 180,E1 -6058.815,E2 -6058.815} C_VEL
LIN {X 0,Y 495.759,Z 95.044,A -85,B 0,C 180,E1 -6061.726,E2 -6061.726} C_VEL
LIN {X 0,Y 495.771,Z 95.038,A -85,B 0,C 180,E1 -6064.694,E2 -6064.694} C_VEL
LIN {X 0,Y 495.731,Z 95.049,A -85,B 0,C 180,E1 -6067.562,E2 -6067.562} C_VEL
LIN {X 0,Y 495.769,Z 95.039,A -85,B 0,C 180,E1 -6070.7,E2 -6070.7} C_VEL
LIN {X 0,Y 495.737,Z 95.042,A -85,B 0,C 180,E1 -6074.001,E2 -6074.001} C_VEL
LIN {X 0,Y 495.728,Z 95.05,A -85,B 0,C 180,E1 -6077.117,E2 -6077.117} C_VEL
LIN {X 0,Y 495.761,Z 95.039,A -85,B 0,C 180,E1 -6079.953,E2 -6079.953} C_VEL
LIN {X 0,Y 495.732,Z 95.044,A -85,B 0,C 180,E1 -6082.553,E2 -6082.553} C_VEL
LIN {X 0,Y 495.785,Z 95.04,A -85,B 0,C 180,E1 -6085.457,E2 -6085.457} C_VEL
LIN {X 0,Y 495.759,Z 95.043,A -85,B 0,C 180,E1 -6088.364,E2 -6088.364} C_VEL
LIN {X 0,Y 495.791,Z 95.041,A -85,B 0,C 180,E1 -6091.507,E2 -6091.507} C_VEL
LIN {X 0,Y 495.818,Z 95.039,A -85,B 0,C 180,E1 -6092.564,E2 -6092.564} C_VEL
LIN {X 0,Y 496.952,Z 98.11,A -85,B 0,C 180,E1 -6092.695,E2 -6092.695} C_VEL
LIN {X 0,Y 505.008,Z 114.568,A -85,B 0,C 180,E1 -6093.443,E2 -6093.443} C_VEL
LIN {X 0,Y 503.168,Z 239.072,A -85,B 0,C 180,E1 -6095.465,E2 -6095.465} C_VEL
LIN {X 0,Y 502.48,Z 291.493,A -85,B 0,C 180,E1 -6096.317,E2 -6096.317} C_VEL
LIN {X 0,Y 502.093,Z 307.58,A -85,B 0,C 180,E1 -6096.735,E2 -6096.735} C_VEL
LIN {X 0,Y 501.607,Z 322.963,A -85,B 0,C 180,E1 -6097.283,E2 -6097.283} C_VEL
LIN {X 0,Y 501.021,Z 338.63,A -85,B 0,C 180,E1 -6098.001,E2 -6098.001} C_VEL
LIN {X 0,Y 500.348,Z 352.784,A -85,B 0,C 180,E1 -6098.796,E2 -6098.796} C_VEL
LIN {X 0,Y 499.572,Z 367.952,A -85,B 0,C 180,E1 -6099.839,E2 -6099.839} C_VEL
LIN {X 0,Y 498.804,Z 381.712,A -85,B 0,C 180,E1 -6100.975,E2 -6100.975} C_VEL
LIN {X 0,Y 498.135,Z 393.62,A -85,B 0,C 180,E1 -6102.13,E2 -6102.13} C_VEL
LIN {X 0,Y 497.529,Z 404.759,A -85,B 0,C 180,E1 -6103.378,E2 -6103.378} C_VEL
LIN {X 0,Y 496.931,Z 415.77,A -85,B 0,C 180,E1 -6104.832,E2 -6104.832} C_VEL
LIN {X 0,Y 496.407,Z 425.162,A -85,B 0,C 180,E1 -6106.282,E2 -6106.282} C_VEL
LIN {X 0,Y 496.012,Z 433.939,A -85,B 0,C 180,E1 -6107.869,E2 -6107.869} C_VEL
LIN {X 0,Y 495.637,Z 440.962,A -85,B 0,C 180,E1 -6109.377,E2 -6109.377} C_VEL
LIN {X 0,Y 495.432,Z 447.324,A -85,B 0,C 180,E1 -6111.023,E2 -6111.023} C_VEL
LIN {X 0,Y 495.306,Z 452.53,A -85,B 0,C 180,E1 -6112.663,E2 -6112.663} C_VEL
LIN {X 0,Y 495.162,Z 456.526,A -85,B 0,C 180,E1 -6114.298,E2 -6114.298} C_VEL
LIN {X 0,Y 495.125,Z 459.539,A -85,B 0,C 180,E1 -6115.93,E2 -6115.93} C_VEL
LIN {X 0,Y 495.058,Z 461.515,A -85,B 0,C 180,E1 -6117.559,E2 -6117.559} C_VEL
LIN {X 0,Y 494.951,Z 462.562,A -85,B 0,C 180,E1 -6119.186,E2 -6119.186} C_VEL
LIN {X 0,Y 494.954,Z 462.626,A -85,B 0,C 180,E1 -6120.813,E2 -6120.813} C_VEL
LIN {X 0,Y 495.059,Z 461.741,A -85,B 0,C 180,E1 -6122.441,E2 -6122.441} C_VEL
LIN {X 0,Y 495.141,Z 459.889,A -85,B 0,C 180,E1 -6124.07,E2 -6124.07} C_VEL
LIN {X 0,Y 495.166,Z 457.03,A -85,B 0,C 180,E1 -6125.702,E2 -6125.702} C_VEL
LIN {X 0,Y 495.35,Z 453.152,A -85,B 0,C 180,E1 -6127.336,E2 -6127.336} C_VEL
LIN {X 0,Y 495.46,Z 448.098,A -85,B 0,C 180,E1 -6128.977,E2 -6128.977} C_VEL
LIN {X 0,Y 495.678,Z 441.875,A -85,B 0,C 180,E1 -6130.621,E2 -6130.621} C_VEL
LIN {X 0,Y 496.074,Z 434.285,A -85,B 0,C 180,E1 -6132.269,E2 -6132.269} C_VEL
LIN {X 0,Y 496.514,Z 425.072,A -85,B 0,C 180,E1 -6133.924,E2 -6133.924} C_VEL
LIN {X 0,Y 497.041,Z 415.496,A -85,B 0,C 180,E1 -6135.374,E2 -6135.374} C_VEL
LIN {X 0,Y 497.656,Z 404.256,A -85,B 0,C 180,E1 -6136.828,E2 -6136.828} C_VEL
LIN {X 0,Y 498.317,Z 391.906,A -85,B 0,C 180,E1 -6138.182,E2 -6138.182} C_VEL
LIN {X 0,Y 499.079,Z 378.274,A -85,B 0,C 180,E1 -6139.44,E2 -6139.44} C_VEL
LIN {X 0,Y 499.802,Z 363.423,A -85,B 0,C 180,E1 -6140.581,E2 -6140.581} C_VEL
LIN {X 0,Y 500.5,Z 347.618,A -85,B 0,C 180,E1 -6141.576,E2 -6141.576} C_VEL
LIN {X 0,Y 501.105,Z 332.135,A -85,B 0,C 180,E1 -6142.36,E2 -6142.36} C_VEL
LIN {X 0,Y 501.607,Z 315.579,A -85,B 0,C 180,E1 -6143.016,E2 -6143.016} C_VEL
LIN {X 0,Y 501.983,Z 299.485,A -85,B 0,C 180,E1 -6143.489,E2 -6143.489} C_VEL
LIN {X 0,Y 502.233,Z 282.374,A -85,B 0,C 180,E1 -6143.832,E2 -6143.832} C_VEL
LIN {X 0,Y 503.858,Z 188.675,A -85,B 0,C 180,E1 -6145.426,E2 -6145.426} C_VEL
LIN {X 0,Y 505.702,Z 115.003,A -85,B 0,C 180,E1 -6146.786,E2 -6146.786} C_VEL
LIN {X 0,Y 499.155,Z 102.088,A -85,B 0,C 180,E1 -6147.536,E2 -6147.536} C_VEL
LIN {X 0,Y 495.971,Z 96.253,A -85,B 0,C 180,E1 -6147.917,E2 -6147.917} C_VEL
LIN {X 0,Y 495.733,Z 95.049,A -85,B 0,C 180,E1 -6147.987,E2 -6147.987} C_VEL
LIN {X 0,Y 495.739,Z 95.05,A -85,B 0,C 180,E1 -6150.688,E2 -6150.688} C_VEL
LIN {X 0,Y 495.753,Z 95.045,A -85,B 0,C 180,E1 -6153.565,E2 -6153.565} C_VEL
LIN {X 0,Y 495.718,Z 95.053,A -85,B 0,C 180,E1 -6156.545,E2 -6156.545} C_VEL
LIN {X 0,Y 495.75,Z 95.045,A -85,B 0,C 180,E1 -6159.638,E2 -6159.638} C_VEL
LIN {X 0,Y 495.739,Z 95.049,A -85,B 0,C 180,E1 -6162.506,E2 -6162.506} C_VEL
LIN {X 0,Y 495.739,Z 95.045,A -85,B 0,C 180,E1 -6165.14,E2 -6165.14} C_VEL
LIN {X 0,Y 495.758,Z 95.047,A -85,B 0,C 180,E1 -6168.218,E2 -6168.218} C_VEL
LIN {X 0,Y 495.751,Z 95.047,A -85,B 0,C 180,E1 -6171.408,E2 -6171.408} C_VEL
LIN {X 0,Y 495.749,Z 95.049,A -85,B 0,C 180,E1 -6174.462,E2 -6174.462} C_VEL
LIN {X 0,Y 495.807,Z 95.249,A -85,B 0,C 180,E1 -6176.537,E2 -6176.537} C_VEL
LIN {X 0,Y 500.005,Z 107.462,A -85,B 0,C 180,E1 -6178.212,E2 -6178.212} C_VEL
LIN {X 0,Y 502.753,Z 117.055,A -85,B 0,C 180,E1 -6179.397,E2 -6179.397} C_VEL
LIN {X 0,Y 502.838,Z 120.945,A -85,B 0,C 180,E1 -6179.79,E2 -6179.79} C_VEL
LIN {X 0,Y 501.353,Z 148.876,A -85,B 0,C 180,E1 -6182.379,E2 -6182.379} C_VEL
LIN {X 0,Y 504.125,Z 168.243,A -85,B 0,C 180,E1 -6182.966,E2 -6182.966} C_VEL
LIN {X 0,Y 505.068,Z 177.074,A -85,B 0,C 180,E1 -6183.206,E2 -6183.206} C_VEL
LIN {X 0,Y 502.863,Z 278.318,A -85,B 0,C 180,E1 -6184.99,E2 -6184.99} C_VEL
LIN {X 0,Y 501.666,Z 360.77,A -85,B 0,C 180,E1 -6186.358,E2 -6186.358} C_VEL
LIN {X 0,Y 501.211,Z 377.078,A -85,B 0,C 180,E1 -6186.773,E2 -6186.773} C_VEL
LIN {X 0,Y 500.61,Z 393.498,A -85,B 0,C 180,E1 -6187.344,E2 -6187.344} C_VEL
LIN {X 0,Y 499.985,Z 408.439,A -85,B 0,C 180,E1 -6188.006,E2 -6188.006} C_VEL
LIN {X 0,Y 499.273,Z 424.002,A -85,B 0,C 180,E1 -6188.856,E2 -6188.856} C_VEL
LIN {X 0,Y 498.545,Z 439.715,A -85,B 0,C 180,E1 -6189.902,E2 -6189.902} C_VEL
LIN {X 0,Y 497.803,Z 454.254,A -85,B 0,C 180,E1 -6191.068,E2 -6191.068} C_VEL
LIN {X 0,Y 497.204,Z 467.329,A -85,B 0,C 180,E1 -6192.307,E2 -6192.307} C_VEL
LIN {X 0,Y 496.699,Z 478.733,A -85,B 0,C 180,E1 -6193.561,E2 -6193.561} C_VEL
LIN {X 0,Y 496.201,Z 490.144,A -85,B 0,C 180,E1 -6195.019,E2 -6195.019} C_VEL
LIN {X 0,Y 495.794,Z 501.096,A -85,B 0,C 180,E1 -6196.682,E2 -6196.682} C_VEL
LIN {X 0,Y 495.509,Z 509.836,A -85,B 0,C 180,E1 -6198.269,E2 -6198.269} C_VEL
LIN {X 0,Y 495.305,Z 516.901,A -85,B 0,C 180,E1 -6199.783,E2 -6199.783} C_VEL
LIN {X 0,Y 495.16,Z 523.302,A -85,B 0,C 180,E1 -6201.429,E2 -6201.429} C_VEL
LIN {X 0,Y 495.149,Z 528.375,A -85,B 0,C 180,E1 -6203.07,E2 -6203.07} C_VEL
LIN {X 0,Y 495.109,Z 531.457,A -85,B 0,C 180,E1 -6204.297,E2 -6204.297} C_VEL
LIN {X 0,Y 495.077,Z 534.596,A -85,B 0,C 180,E1 -6205.929,E2 -6205.929} C_VEL
LIN {X 0,Y 495.052,Z 536.656,A -85,B 0,C 180,E1 -6207.559,E2 -6207.559} C_VEL
LIN {X 0,Y 494.928,Z 537.691,A -85,B 0,C 180,E1 -6209.186,E2 -6209.186} C_VEL
LIN {X 0,Y 494.925,Z 537.728,A -85,B 0,C 180,E1 -6210.813,E2 -6210.813} C_VEL
LIN {X 0,Y 495.048,Z 536.761,A -85,B 0,C 180,E1 -6212.44,E2 -6212.44} C_VEL
LIN {X 0,Y 495.075,Z 534.782,A -85,B 0,C 180,E1 -6214.07,E2 -6214.07} C_VEL
LIN {X 0,Y 495.084,Z 531.734,A -85,B 0,C 180,E1 -6215.702,E2 -6215.702} C_VEL
LIN {X 0,Y 495.14,Z 527.638,A -85,B 0,C 180,E1 -6217.339,E2 -6217.339} C_VEL
LIN {X 0,Y 495.194,Z 522.315,A -85,B 0,C 180,E1 -6218.981,E2 -6218.981} C_VEL
LIN {X 0,Y 495.347,Z 515.801,A -85,B 0,C 180,E1 -6220.628,E2 -6220.628} C_VEL
LIN {X 0,Y 495.642,Z 507.894,A -85,B 0,C 180,E1 -6222.28,E2 -6222.28} C_VEL
LIN {X 0,Y 495.948,Z 498.363,A -85,B 0,C 180,E1 -6223.939,E2 -6223.939} C_VEL
LIN {X 0,Y 496.393,Z 488.541,A -85,B 0,C 180,E1 -6225.394,E2 -6225.394} C_VEL
LIN {X 0,Y 496.958,Z 477.065,A -85,B 0,C 180,E1 -6226.852,E2 -6226.852} C_VEL
LIN {X 0,Y 497.653,Z 464.564,A -85,B 0,C 180,E1 -6228.207,E2 -6228.207} C_VEL
LIN {X 0,Y 498.371,Z 451.25,A -85,B 0,C 180,E1 -6229.428,E2 -6229.428} C_VEL
LIN {X 0,Y 499.098,Z 437.436,A -85,B 0,C 180,E1 -6230.503,E2 -6230.503} C_VEL
LIN {X 0,Y 499.85,Z 423.143,A -85,B 0,C 180,E1 -6231.442,E2 -6231.442} C_VEL
LIN {X 0,Y 500.588,Z 407.805,A -85,B 0,C 180,E1 -6232.275,E2 -6232.275} C_VEL
LIN {X 0,Y 501.354,Z 390.82,A -85,B 0,C 180,E1 -6233.001,E2 -6233.001} C_VEL
LIN {X 0,Y 501.986,Z 373.703,A -85,B 0,C 180,E1 -6233.543,E2 -6233.543} C_VEL
LIN {X 0,Y 502.413,Z 357.031,A -85,B 0,C 180,E1 -6233.905,E2 -6233.905} C_VEL
LIN {X 0,Y 505.071,Z 176.006,A -85,B 0,C 180,E1 -6236.812,E2 -6236.812} C_VEL
LIN {X 0,Y 501.748,Z 154.321,A -85,B 0,C 180,E1 -6237.384,E2 -6237.384} C_VEL
LIN {X 0,Y 503.128,Z 124.184,A -85,B 0,C 180,E1 -6240.089,E2 -6240.089} C_VEL
LIN {X 0,Y 503.241,Z 118.438,A -85,B 0,C 180,E1 -6240.618,E2 -6240.618} C_VEL
LIN {X 0,Y 496.583,Z 97.558,A -85,B 0,C 180,E1 -6243.022,E2 -6243.022} C_VEL
LIN {X 0,Y 495.78,Z 95.043,A -85,B 0,C 180,E1 -6243.341,E2 -6243.341} C_VEL
LIN {X 0,Y 495.724,Z 95.051,A -85,B 0,C 180,E1 -6246.543,E2 -6246.543} C_VEL
LIN {X 0,Y 495.752,Z 95.043,A -85,B 0,C 180,E1 -6249.638,E2 -6249.638} C_VEL
LIN {X 0,Y 495.777,Z 95.045,A -85,B 0,C 180,E1 -6252.512,E2 -6252.512} C_VEL
LIN {X 0,Y 495.745,Z 95.043,A -85,B 0,C 180,E1 -6255.139,E2 -6255.139} C_VEL
LIN {X 0,Y 495.752,Z 95.046,A -85,B 0,C 180,E1 -6258.219,E2 -6258.219} C_VEL
LIN {X 0,Y 495.747,Z 95.04,A -85,B 0,C 180,E1 -6261.408,E2 -6261.408} C_VEL
LIN {X 0,Y 495.753,Z 95.045,A -85,B 0,C 180,E1 -6264.463,E2 -6264.463} C_VEL
LIN {X 0,Y 495.764,Z 95.038,A -85,B 0,C 180,E1 -6267.406,E2 -6267.406} C_VEL
LIN {X 0,Y 495.763,Z 95.045,A -85,B 0,C 180,E1 -6270.254,E2 -6270.254} C_VEL
LIN {X 0,Y 495.819,Z 95.031,A -85,B 0,C 180,E1 -6273.251,E2 -6273.251} C_VEL
LIN {X 0,Y 495.748,Z 95.044,A -85,B 0,C 180,E1 -6275.725,E2 -6275.725} C_VEL
LIN {X 0,Y 495.74,Z 95.045,A -85,B 0,C 180,E1 -6278.371,E2 -6278.371} C_VEL
LIN {X 0,Y 495.78,Z 95.036,A -85,B 0,C 180,E1 -6280.972,E2 -6280.972} C_VEL
LIN {X 0,Y 495.775,Z 95.04,A -85,B 0,C 180,E1 -6283.53,E2 -6283.53} C_VEL
LIN {X 0,Y 495.79,Z 95.041,A -85,B 0,C 180,E1 -6286.056,E2 -6286.056} C_VEL
LIN {X 0,Y 495.869,Z 95.026,A -85,B 0,C 180,E1 -6288.555,E2 -6288.555} C_VEL
LIN {X 0,Y 495.868,Z 95.033,A -85,B 0,C 180,E1 -6291.852,E2 -6291.852} C_VEL
LIN {X 0,Y 495.891,Z 95.024,A -85,B 0,C 180,E1 -6294.307,E2 -6294.307} C_VEL
LIN {X 0,Y 495.989,Z 95.017,A -85,B 0,C 180,E1 -6297.564,E2 -6297.564} C_VEL
LIN {X 0,Y 495.994,Z 95.013,A -85,B 0,C 180,E1 -6300,E2 -6300} C_VEL
LIN {X 0,Y 495.989,Z 95.01,A -85,B 0,C 180,E1 -6302.436,E2 -6302.436} C_VEL
LIN {X 0,Y 495.891,Z 95.029,A -85,B 0,C 180,E1 -6305.694,E2 -6305.694} C_VEL
LIN {X 0,Y 495.868,Z 95.026,A -85,B 0,C 180,E1 -6308.148,E2 -6308.148} C_VEL
LIN {X 0,Y 495.847,Z 95.036,A -85,B 0,C 180,E1 -6311.445,E2 -6311.445} C_VEL
LIN {X 0,Y 495.786,Z 95.037,A -85,B 0,C 180,E1 -6314.783,E2 -6314.783} C_VEL
LIN {X 0,Y 495.783,Z 95.045,A -85,B 0,C 180,E1 -6317.319,E2 -6317.319} C_VEL
LIN {X 0,Y 495.774,Z 95.038,A -85,B 0,C 180,E1 -6319.89,E2 -6319.89} C_VEL
LIN {X 0,Y 495.761,Z 95.042,A -85,B 0,C 180,E1 -6322.863,E2 -6322.863} C_VEL
LIN {X 0,Y 495.787,Z 95.035,A -85,B 0,C 180,E1 -6326.068,E2 -6326.068} C_VEL
LIN {X 0,Y 495.768,Z 95.042,A -85,B 0,C 180,E1 -6328.815,E2 -6328.815} C_VEL
LIN {X 0,Y 495.755,Z 95.04,A -85,B 0,C 180,E1 -6331.726,E2 -6331.726} C_VEL
LIN {X 0,Y 495.773,Z 95.041,A -85,B 0,C 180,E1 -6334.696,E2 -6334.696} C_VEL
LIN {X 0,Y 495.728,Z 95.044,A -85,B 0,C 180,E1 -6337.562,E2 -6337.562} C_VEL
LIN {X 0,Y 495.763,Z 95.044,A -85,B 0,C 180,E1 -6340.7,E2 -6340.7} C_VEL
LIN {X 0,Y 495.731,Z 95.042,A -85,B 0,C 180,E1 -6343.696,E2 -6343.696} C_VEL
LIN {X 0,Y 495.732,Z 95.044,A -85,B 0,C 180,E1 -6346.305,E2 -6346.305} C_VEL
LIN {X 0,Y 495.764,Z 95.04,A -85,B 0,C 180,E1 -6349.301,E2 -6349.301} C_VEL
LIN {X 0,Y 495.727,Z 95.047,A -85,B 0,C 180,E1 -6352.439,E2 -6352.439} C_VEL
LIN {X 0,Y 495.775,Z 95.037,A -85,B 0,C 180,E1 -6355.457,E2 -6355.457} C_VEL
LIN {X 0,Y 495.754,Z 95.044,A -85,B 0,C 180,E1 -6358.364,E2 -6358.364} C_VEL
LIN {X 0,Y 495.751,Z 95.04,A -85,B 0,C 180,E1 -6360.759,E2 -6360.759} C_VEL
LIN {X 0,Y 495.094,Z 95.124,A -85,B 0,C 180,E1 -6361.438,E2 -6361.438} C_VEL
LIN {X 0,Y 492.237,Z 95.486,A -85,B 0,C 180,E1 -6362.54,E2 -6362.54} C_VEL
LIN {X 0,Y 489.829,Z 95.781,A -85,B 0,C 180,E1 -6363.429,E2 -6363.429} C_VEL
LIN {X 0,Y 488.813,Z 95.908,A -85,B 0,C 180,E1 -6364.115,E2 -6364.115} C_VEL
LIN {X 0,Y 488.741,Z 95.919,A -85,B 0,C 180,E1 -6364.348,E2 -6364.348} C_VEL
LIN {X 0,Y 488.723,Z 95.916,A -85,B 0,C 180,E1 -6367.154,E2 -6367.154} C_VEL
LIN {X 0,Y 488.724,Z 95.916,A -85,B 0,C 180,E1 -6369.811,E2 -6369.811} C_VEL
LIN {X 0,Y 488.734,Z 95.922,A -85,B 0,C 180,E1 -6372.424,E2 -6372.424} C_VEL
LIN {X 0,Y 488.762,Z 95.911,A -85,B 0,C 180,E1 -6375,E2 -6375} C_VEL
LIN {X 0,Y 488.805,Z 95.912,A -85,B 0,C 180,E1 -6378.388,E2 -6378.388} C_VEL
LIN {X 0,Y 488.817,Z 95.906,A -85,B 0,C 180,E1 -6381.734,E2 -6381.734} C_VEL
LIN {X 0,Y 488.855,Z 95.907,A -85,B 0,C 180,E1 -6384.225,E2 -6384.225} C_VEL
LIN {X 0,Y 488.962,Z 95.887,A -85,B 0,C 180,E1 -6387.529,E2 -6387.529} C_VEL
LIN {X 0,Y 488.935,Z 95.889,A -85,B 0,C 180,E1 -6390.824,E2 -6390.824} C_VEL
LIN {X 0,Y 488.962,Z 95.888,A -85,B 0,C 180,E1 -6392.472,E2 -6392.472} C_VEL
LIN {X 0,Y 488.855,Z 95.905,A -85,B 0,C 180,E1 -6395.776,E2 -6395.776} C_VEL
LIN {X 0,Y 488.819,Z 95.907,A -85,B 0,C 180,E1 -6398.267,E2 -6398.267} C_VEL
LIN {X 0,Y 488.807,Z 95.91,A -85,B 0,C 180,E1 -6401.613,E2 -6401.613} C_VEL
LIN {X 0,Y 488.764,Z 95.91,A -85,B 0,C 180,E1 -6405.001,E2 -6405.001} C_VEL
LIN {X 0,Y 488.757,Z 95.912,A -85,B 0,C 180,E1 -6408.443,E2 -6408.443} C_VEL
LIN {X 0,Y 488.709,Z 95.918,A -85,B 0,C 180,E1 -6411.071,E2 -6411.071} C_VEL
LIN {X 0,Y 488.682,Z 95.927,A -85,B 0,C 180,E1 -6413.747,E2 -6413.747} C_VEL
LIN {X 0,Y 488.794,Z 95.907,A -85,B 0,C 180,E1 -6416.944,E2 -6416.944} C_VEL
LIN {X 0,Y 488.712,Z 95.917,A -85,B 0,C 180,E1 -6420.363,E2 -6420.363} C_VEL
LIN {X 0,Y 488.737,Z 95.922,A -85,B 0,C 180,E1 -6423.485,E2 -6423.485} C_VEL
LIN {X 0,Y 488.684,Z 95.92,A -85,B 0,C 180,E1 -6426.355,E2 -6426.355} C_VEL
LIN {X 0,Y 488.703,Z 95.925,A -85,B 0,C 180,E1 -6429.255,E2 -6429.255} C_VEL
LIN {X 0,Y 488.71,Z 95.922,A -85,B 0,C 180,E1 -6431.6,E2 -6431.6} C_VEL
LIN {X 0,Y 488.715,Z 95.919,A -85,B 0,C 180,E1 -6434.802,E2 -6434.802} C_VEL
LIN {X 0,Y 488.694,Z 95.924,A -85,B 0,C 180,E1 -6437.475,E2 -6437.475} C_VEL
LIN {X 0,Y 488.736,Z 95.916,A -85,B 0,C 180,E1 -6439.677,E2 -6439.677} C_VEL
LIN {X 0,Y 488.683,Z 95.925,A -85,B 0,C 180,E1 -6442.841,E2 -6442.841} C_VEL
LIN {X 0,Y 488.736,Z 95.915,A -85,B 0,C 180,E1 -6445.888,E2 -6445.888} C_VEL
LIN {X 0,Y 488.696,Z 95.925,A -85,B 0,C 180,E1 -6448.821,E2 -6448.821} C_VEL
LIN {X 0,Y 488.757,Z 95.916,A -85,B 0,C 180,E1 -6452.159,E2 -6452.159} C_VEL
LIN {X 0,Y 489.927,Z 99.033,A -85,B 0,C 180,E1 -6452.3,E2 -6452.3} C_VEL
LIN {X 0,Y 498.576,Z 116.561,A -85,B 0,C 180,E1 -6453.118,E2 -6453.118} C_VEL
LIN {X 0,Y 497.232,Z 198.966,A -85,B 0,C 180,E1 -6454.491,E2 -6454.491} C_VEL
LIN {X 0,Y 495.893,Z 291.385,A -85,B 0,C 180,E1 -6456.01,E2 -6456.01} C_VEL
LIN {X 0,Y 495.497,Z 307.563,A -85,B 0,C 180,E1 -6456.434,E2 -6456.434} C_VEL
LIN {X 0,Y 494.959,Z 323.694,A -85,B 0,C 180,E1 -6457.016,E2 -6457.016} C_VEL
LIN {X 0,Y 494.374,Z 338.259,A -85,B 0,C 180,E1 -6457.688,E2 -6457.688} C_VEL
LIN {X 0,Y 493.664,Z 352.536,A -85,B 0,C 180,E1 -6458.495,E2 -6458.495} C_VEL
LIN {X 0,Y 492.814,Z 367.829,A -85,B 0,C 180,E1 -6459.55,E2 -6459.55} C_VEL
LIN {X 0,Y 492.03,Z 381.12,A -85,B 0,C 180,E1 -6460.649,E2 -6460.649} C_VEL
LIN {X 0,Y 491.323,Z 393.712,A -85,B 0,C 180,E1 -6461.873,E2 -6461.873} C_VEL
LIN {X 0,Y 490.638,Z 404.915,A -85,B 0,C 180,E1 -6463.138,E2 -6463.138} C_VEL
LIN {X 0,Y 490.013,Z 415.998,A -85,B 0,C 180,E1 -6464.613,E2 -6464.613} C_VEL
LIN {X 0,Y 489.446,Z 425.458,A -85,B 0,C 180,E1 -6466.083,E2 -6466.083} C_VEL
LIN {X 0,Y 489.002,Z 434.661,A -85,B 0,C 180,E1 -6467.772,E2 -6467.772} C_VEL
LIN {X 0,Y 488.546,Z 443.078,A -85,B 0,C 180,E1 -6469.641,E2 -6469.641} C_VEL
LIN {X 0,Y 488.356,Z 449.171,A -85,B 0,C 180,E1 -6471.309,E2 -6471.309} C_VEL
LIN {X 0,Y 488.239,Z 454.048,A -85,B 0,C 180,E1 -6472.972,E2 -6472.972} C_VEL
LIN {X 0,Y 488.11,Z 457.001,A -85,B 0,C 180,E1 -6474.215,E2 -6474.215} C_VEL
LIN {X 0,Y 488.061,Z 460.04,A -85,B 0,C 180,E1 -6475.871,E2 -6475.871} C_VEL
LIN {X 0,Y 487.997,Z 462.035,A -85,B 0,C 180,E1 -6477.524,E2 -6477.524} C_VEL
LIN {X 0,Y 487.872,Z 463.096,A -85,B 0,C 180,E1 -6479.175,E2 -6479.175} C_VEL
LIN {X 0,Y 487.876,Z 463.171,A -85,B 0,C 180,E1 -6480.825,E2 -6480.825} C_VEL
LIN {X 0,Y 487.998,Z 462.284,A -85,B 0,C 180,E1 -6482.476,E2 -6482.476} C_VEL
LIN {X 0,Y 488.079,Z 460.432,A -85,B 0,C 180,E1 -6484.129,E2 -6484.129} C_VEL
LIN {X 0,Y 488.116,Z 457.56,A -85,B 0,C 180,E1 -6485.784,E2 -6485.784} C_VEL
LIN {X 0,Y 488.308,Z 453.673,A -85,B 0,C 180,E1 -6487.442,E2 -6487.442} C_VEL
LIN {X 0,Y 488.515,Z 447.194,A -85,B 0,C 180,E1 -6489.523,E2 -6489.523} C_VEL
LIN {X 0,Y 488.819,Z 440.552,A -85,B 0,C 180,E1 -6491.192,E2 -6491.192} C_VEL
LIN {X 0,Y 489.208,Z 432.528,A -85,B 0,C 180,E1 -6492.866,E2 -6492.866} C_VEL
LIN {X 0,Y 489.742,Z 422.886,A -85,B 0,C 180,E1 -6494.544,E2 -6494.544} C_VEL
LIN {X 0,Y 490.341,Z 412.739,A -85,B 0,C 180,E1 -6496.035,E2 -6496.035} C_VEL
LIN {X 0,Y 491.023,Z 401.011,A -85,B 0,C 180,E1 -6497.492,E2 -6497.492} C_VEL
LIN {X 0,Y 491.747,Z 387.883,A -85,B 0,C 180,E1 -6498.866,E2 -6498.866} C_VEL
LIN {X 0,Y 492.543,Z 374.693,A -85,B 0,C 180,E1 -6500.026,E2 -6500.026} C_VEL
LIN {X 0,Y 493.261,Z 360.405,A -85,B 0,C 180,E1 -6501.085,E2 -6501.085} C_VEL
LIN {X 0,Y 494.014,Z 345.237,A -85,B 0,C 180,E1 -6502.012,E2 -6502.012} C_VEL
LIN {X 0,Y 494.639,Z 329.766,A -85,B 0,C 180,E1 -6502.779,E2 -6502.779} C_VEL
LIN {X 0,Y 495.113,Z 313.143,A -85,B 0,C 180,E1 -6503.419,E2 -6503.419} C_VEL
LIN {X 0,Y 495.477,Z 296.871,A -85,B 0,C 180,E1 -6503.872,E2 -6503.872} C_VEL
LIN {X 0,Y 495.883,Z 274.179,A -85,B 0,C 180,E1 -6504.288,E2 -6504.288} C_VEL
LIN {X 0,Y 497.663,Z 185.972,A -85,B 0,C 180,E1 -6505.85,E2 -6505.85} C_VEL
LIN {X 0,Y 499.593,Z 117.313,A -85,B 0,C 180,E1 -6507.165,E2 -6507.165} C_VEL
LIN {X 0,Y 493.21,Z 104.783,A -85,B 0,C 180,E1 -6507.935,E2 -6507.935} C_VEL
LIN {X 0,Y 490.185,Z 99.472,A -85,B 0,C 180,E1 -6508.315,E2 -6508.315} C_VEL
LIN {X 0,Y 488.867,Z 96.8,A -85,B 0,C 180,E1 -6508.488,E2 -6508.488} C_VEL
LIN {X 0,Y 488.697,Z 95.925,A -85,B 0,C 180,E1 -6508.527,E2 -6508.527} C_VEL
LIN {X 0,Y 488.684,Z 95.928,A -85,B 0,C 180,E1 -6511.18,E2 -6511.18} C_VEL
LIN {X 0,Y 488.725,Z 95.922,A -85,B 0,C 180,E1 -6514.113,E2 -6514.113} C_VEL
LIN {X 0,Y 488.671,Z 95.928,A -85,B 0,C 180,E1 -6517.159,E2 -6517.159} C_VEL
LIN {X 0,Y 488.72,Z 95.923,A -85,B 0,C 180,E1 -6520.344,E2 -6520.344} C_VEL
LIN {X 0,Y 488.686,Z 95.925,A -85,B 0,C 180,E1 -6523.654,E2 -6523.654} C_VEL
LIN {X 0,Y 488.686,Z 95.928,A -85,B 0,C 180,E1 -6526.345,E2 -6526.345} C_VEL
LIN {X 0,Y 488.735,Z 95.921,A -85,B 0,C 180,E1 -6529.676,E2 -6529.676} C_VEL
LIN {X 0,Y 488.68,Z 95.927,A -85,B 0,C 180,E1 -6532.841,E2 -6532.841} C_VEL
LIN {X 0,Y 488.74,Z 96.044,A -85,B 0,C 180,E1 -6535.954,E2 -6535.954} C_VEL
LIN {X 0,Y 492.822,Z 107.471,A -85,B 0,C 180,E1 -6537.626,E2 -6537.626} C_VEL
LIN {X 0,Y 496.349,Z 119.629,A -85,B 0,C 180,E1 -6539.197,E2 -6539.197} C_VEL
LIN {X 0,Y 496.362,Z 123.176,A -85,B 0,C 180,E1 -6539.563,E2 -6539.563} C_VEL
LIN {X 0,Y 494.883,Z 147.67,A -85,B 0,C 180,E1 -6541.892,E2 -6541.892} C_VEL
LIN {X 0,Y 497.819,Z 168.032,A -85,B 0,C 180,E1 -6542.544,E2 -6542.544} C_VEL
LIN {X 0,Y 498.847,Z 177.784,A -85,B 0,C 180,E1 -6542.823,E2 -6542.823} C_VEL
LIN {X 0,Y 496.433,Z 275.913,A -85,B 0,C 180,E1 -6544.615,E2 -6544.615} C_VEL
LIN {X 0,Y 495.022,Z 360.971,A -85,B 0,C 180,E1 -6546.076,E2 -6546.076} C_VEL
LIN {X 0,Y 494.49,Z 377.874,A -85,B 0,C 180,E1 -6546.521,E2 -6546.521} C_VEL
LIN {X 0,Y 493.763,Z 395.806,A -85,B 0,C 180,E1 -6547.178,E2 -6547.178} C_VEL
LIN {X 0,Y 492.97,Z 412.756,A -85,B 0,C 180,E1 -6547.989,E2 -6547.989} C_VEL
LIN {X 0,Y 492.238,Z 427.597,A -85,B 0,C 180,E1 -6548.868,E2 -6548.868} C_VEL
LIN {X 0,Y 491.474,Z 442.545,A -85,B 0,C 180,E1 -6549.928,E2 -6549.928} C_VEL
LIN {X 0,Y 490.664,Z 457.099,A -85,B 0,C 180,E1 -6551.157,E2 -6551.157} C_VEL
LIN {X 0,Y 490.05,Z 470.278,A -85,B 0,C 180,E1 -6552.472,E2 -6552.472} C_VEL
LIN {X 0,Y 489.446,Z 482.881,A -85,B 0,C 180,E1 -6553.953,E2 -6553.953} C_VEL
LIN {X 0,Y 489.041,Z 493.538,A -85,B 0,C 180,E1 -6555.434,E2 -6555.434} C_VEL
LIN {X 0,Y 488.645,Z 502.653,A -85,B 0,C 180,E1 -6556.907,E2 -6556.907} C_VEL
LIN {X 0,Y 488.392,Z 510.482,A -85,B 0,C 180,E1 -6558.377,E2 -6558.377} C_VEL
LIN {X 0,Y 488.159,Z 517.897,A -85,B 0,C 180,E1 -6560.051,E2 -6560.051} C_VEL
LIN {X 0,Y 488.077,Z 523.998,A -85,B 0,C 180,E1 -6561.72,E2 -6561.72} C_VEL
LIN {X 0,Y 488.074,Z 529.186,A -85,B 0,C 180,E1 -6563.493,E2 -6563.493} C_VEL
LIN {X 0,Y 487.926,Z 532.549,A -85,B 0,C 180,E1 -6565.042,E2 -6565.042} C_VEL
LIN {X 0,Y 487.984,Z 535.228,A -85,B 0,C 180,E1 -6566.697,E2 -6566.697} C_VEL
LIN {X 0,Y 487.892,Z 536.737,A -85,B 0,C 180,E1 -6568.349,E2 -6568.349} C_VEL
LIN {X 0,Y 487.844,Z 537.339,A -85,B 0,C 180,E1 -6569.999,E2 -6569.999} C_VEL
LIN {X 0,Y 487.89,Z 536.827,A -85,B 0,C 180,E1 -6571.65,E2 -6571.65} C_VEL
LIN {X 0,Y 487.964,Z 535.399,A -85,B 0,C 180,E1 -6573.302,E2 -6573.302} C_VEL
LIN {X 0,Y 487.918,Z 532.837,A -85,B 0,C 180,E1 -6574.957,E2 -6574.957} C_VEL
LIN {X 0,Y 488.035,Z 529.286,A -85,B 0,C 180,E1 -6576.615,E2 -6576.615} C_VEL
LIN {X 0,Y 488.076,Z 524.551,A -85,B 0,C 180,E1 -6578.278,E2 -6578.278} C_VEL
LIN {X 0,Y 488.155,Z 518.622,A -85,B 0,C 180,E1 -6579.948,E2 -6579.948} C_VEL
LIN {X 0,Y 488.399,Z 511.426,A -85,B 0,C 180,E1 -6581.622,E2 -6581.622} C_VEL
LIN {X 0,Y 488.719,Z 502.687,A -85,B 0,C 180,E1 -6583.302,E2 -6583.302} C_VEL
LIN {X 0,Y 489.161,Z 493.648,A -85,B 0,C 180,E1 -6584.774,E2 -6584.774} C_VEL
LIN {X 0,Y 489.698,Z 483.141,A -85,B 0,C 180,E1 -6586.251,E2 -6586.251} C_VEL
LIN {X 0,Y 490.339,Z 470.779,A -85,B 0,C 180,E1 -6587.732,E2 -6587.732} C_VEL
LIN {X 0,Y 491.082,Z 457.564,A -85,B 0,C 180,E1 -6589.07,E2 -6589.07} C_VEL
LIN {X 0,Y 491.916,Z 443.515,A -85,B 0,C 180,E1 -6590.27,E2 -6590.27} C_VEL
LIN {X 0,Y 492.721,Z 428.766,A -85,B 0,C 180,E1 -6591.328,E2 -6591.328} C_VEL
LIN {X 0,Y 493.575,Z 413.166,A -85,B 0,C 180,E1 -6592.252,E2 -6592.252} C_VEL
LIN {X 0,Y 494.312,Z 398.52,A -85,B 0,C 180,E1 -6592.96,E2 -6592.96} C_VEL
LIN {X 0,Y 495.061,Z 380.96,A -85,B 0,C 180,E1 -6593.615,E2 -6593.615} C_VEL
LIN {X 0,Y 495.612,Z 364.209,A -85,B 0,C 180,E1 -6594.059,E2 -6594.059} C_VEL
LIN {X 0,Y 496.159,Z 332.139,A -85,B 0,C 180,E1 -6594.601,E2 -6594.601} C_VEL
LIN {X 0,Y 498.639,Z 176.259,A -85,B 0,C 180,E1 -6597.164,E2 -6597.164} C_VEL
LIN {X 0,Y 495.184,Z 153.992,A -85,B 0,C 180,E1 -6597.766,E2 -6597.766} C_VEL
LIN {X 0,Y 496.715,Z 122.548,A -85,B 0,C 180,E1 -6600.621,E2 -6600.621} C_VEL
LIN {X 0,Y 496.761,Z 121.104,A -85,B 0,C 180,E1 -6600.754,E2 -6600.754} C_VEL
LIN {X 0,Y 490.273,Z 100.664,A -85,B 0,C 180,E1 -6603.134,E2 -6603.134} C_VEL
LIN {X 0,Y 488.728,Z 95.921,A -85,B 0,C 180,E1 -6603.716,E2 -6603.716} C_VEL
LIN {X 0,Y 488.678,Z 95.928,A -85,B 0,C 180,E1 -6606.354,E2 -6606.354} C_VEL
LIN {X 0,Y 488.696,Z 95.922,A -85,B 0,C 180,E1 -6609.254,E2 -6609.254} C_VEL
LIN {X 0,Y 488.731,Z 95.923,A -85,B 0,C 180,E1 -6612.52,E2 -6612.52} C_VEL
LIN {X 0,Y 488.708,Z 95.92,A -85,B 0,C 180,E1 -6615.198,E2 -6615.198} C_VEL
LIN {X 0,Y 488.703,Z 95.926,A -85,B 0,C 180,E1 -6618.4,E2 -6618.4} C_VEL
LIN {X 0,Y 488.7,Z 95.919,A -85,B 0,C 180,E1 -6620.947,E2 -6620.947} C_VEL
LIN {X 0,Y 488.681,Z 95.924,A -85,B 0,C 180,E1 -6623.868,E2 -6623.868} C_VEL
LIN {X 0,Y 488.734,Z 95.915,A -85,B 0,C 180,E1 -6626.877,E2 -6626.877} C_VEL
LIN {X 0,Y 488.721,Z 95.919,A -85,B 0,C 180,E1 -6629.781,E2 -6629.781} C_VEL
LIN {X 0,Y 488.787,Z 95.907,A -85,B 0,C 180,E1 -6633.056,E2 -6633.056} C_VEL
LIN {X 0,Y 488.69,Z 95.925,A -85,B 0,C 180,E1 -6636.255,E2 -6636.255} C_VEL
LIN {X 0,Y 488.741,Z 95.913,A -85,B 0,C 180,E1 -6639.176,E2 -6639.176} C_VEL
LIN {X 0,Y 488.729,Z 95.917,A -85,B 0,C 180,E1 -6642.423,E2 -6642.423} C_VEL
LIN {X 0,Y 488.758,Z 95.911,A -85,B 0,C 180,E1 -6645,E2 -6645} C_VEL
LIN {X 0,Y 488.828,Z 95.904,A -85,B 0,C 180,E1 -6648.388,E2 -6648.388} C_VEL
LIN {X 0,Y 488.813,Z 95.912,A -85,B 0,C 180,E1 -6651.734,E2 -6651.734} C_VEL
LIN {X 0,Y 488.85,Z 95.902,A -85,B 0,C 180,E1 -6654.224,E2 -6654.224} C_VEL
LIN {X 0,Y 488.957,Z 95.893,A -85,B 0,C 180,E1 -6657.529,E2 -6657.529} C_VEL
LIN {X 0,Y 488.95,Z 95.887,A -85,B 0,C 180,E1 -6660.824,E2 -6660.824} C_VEL
LIN {X 0,Y 488.957,Z 95.886,A -85,B 0,C 180,E1 -6662.471,E2 -6662.471} C_VEL
LIN {X 0,Y 488.85,Z 95.904,A -85,B 0,C 180,E1 -6665.776,E2 -6665.776} C_VEL
LIN {X 0,Y 488.813,Z 95.904,A -85,B 0,C 180,E1 -6668.267,E2 -6668.267} C_VEL
LIN {X 0,Y 488.801,Z 95.911,A -85,B 0,C 180,E1 -6671.613,E2 -6671.613} C_VEL
LIN {X 0,Y 488.758,Z 95.914,A -85,B 0,C 180,E1 -6675.001,E2 -6675.001} C_VEL
LIN {X 0,Y 488.751,Z 95.912,A -85,B 0,C 180,E1 -6678.442,E2 -6678.442} C_VEL
LIN {X 0,Y 488.703,Z 95.923,A -85,B 0,C 180,E1 -6681.071,E2 -6681.071} C_VEL
LIN {X 0,Y 488.689,Z 95.921,A -85,B 0,C 180,E1 -6683.746,E2 -6683.746} C_VEL
LIN {X 0,Y 488.788,Z 95.913,A -85,B 0,C 180,E1 -6686.944,E2 -6686.944} C_VEL
LIN {X 0,Y 488.706,Z 95.918,A -85,B 0,C 180,E1 -6690.363,E2 -6690.363} C_VEL
LIN {X 0,Y 488.732,Z 95.917,A -85,B 0,C 180,E1 -6693.485,E2 -6693.485} C_VEL
LIN {X 0,Y 488.685,Z 95.921,A -85,B 0,C 180,E1 -6696.356,E2 -6696.356} C_VEL
LIN {X 0,Y 488.698,Z 95.922,A -85,B 0,C 180,E1 -6699.255,E2 -6699.255} C_VEL
LIN {X 0,Y 488.72,Z 95.916,A -85,B 0,C 180,E1 -6701.602,E2 -6701.602} C_VEL
LIN {X 0,Y 488.709,Z 95.925,A -85,B 0,C 180,E1 -6704.802,E2 -6704.802} C_VEL
LIN {X 0,Y 488.692,Z 95.92,A -85,B 0,C 180,E1 -6707.475,E2 -6707.475} C_VEL
LIN {X 0,Y 488.727,Z 95.924,A -85,B 0,C 180,E1 -6710.749,E2 -6710.749} C_VEL
LIN {X 0,Y 488.674,Z 95.921,A -85,B 0,C 180,E1 -6713.868,E2 -6713.868} C_VEL
LIN {X 0,Y 488.736,Z 95.919,A -85,B 0,C 180,E1 -6716.878,E2 -6716.878} C_VEL
LIN {X 0,Y 488.722,Z 95.916,A -85,B 0,C 180,E1 -6719.781,E2 -6719.781} C_VEL
LIN {X 0,Y 488.79,Z 95.909,A -85,B 0,C 180,E1 -6723.057,E2 -6723.057} C_VEL
LIN {X 0,Y 488.741,Z 95.919,A -85,B 0,C 180,E1 -6724.348,E2 -6724.348} C_VEL
LIN {X 0,Y 488.097,Z 96.006,A -85,B 0,C 180,E1 -6725.036,E2 -6725.036} C_VEL
LIN {X 0,Y 485.228,Z 96.361,A -85,B 0,C 180,E1 -6726.152,E2 -6726.152} C_VEL
LIN {X 0,Y 482.781,Z 96.658,A -85,B 0,C 180,E1 -6727.052,E2 -6727.052} C_VEL
LIN {X 0,Y 481.723,Z 96.788,A -85,B 0,C 180,E1 -6727.747,E2 -6727.747} C_VEL
LIN {X 0,Y 481.635,Z 96.799,A -85,B 0,C 180,E1 -6727.983,E2 -6727.983} C_VEL
LIN {X 0,Y 481.705,Z 96.798,A -85,B 0,C 180,E1 -6730.394,E2 -6730.394} C_VEL
LIN {X 0,Y 481.69,Z 96.792,A -85,B 0,C 180,E1 -6733.035,E2 -6733.035} C_VEL
LIN {X 0,Y 481.689,Z 96.792,A -85,B 0,C 180,E1 -6735.639,E2 -6735.639} C_VEL
LIN {X 0,Y 481.751,Z 96.792,A -85,B 0,C 180,E1 -6738.216,E2 -6738.216} C_VEL
LIN {X 0,Y 481.763,Z 96.784,A -85,B 0,C 180,E1 -6741.612,E2 -6741.612} C_VEL
LIN {X 0,Y 481.816,Z 96.784,A -85,B 0,C 180,E1 -6744.14,E2 -6744.14} C_VEL
LIN {X 0,Y 481.928,Z 96.763,A -85,B 0,C 180,E1 -6747.493,E2 -6747.493} C_VEL
LIN {X 0,Y 481.887,Z 96.767,A -85,B 0,C 180,E1 -6750.836,E2 -6750.836} C_VEL
LIN {X 0,Y 481.928,Z 96.764,A -85,B 0,C 180,E1 -6752.508,E2 -6752.508} C_VEL
LIN {X 0,Y 481.816,Z 96.783,A -85,B 0,C 180,E1 -6755.861,E2 -6755.861} C_VEL
LIN {X 0,Y 481.764,Z 96.784,A -85,B 0,C 180,E1 -6758.389,E2 -6758.389} C_VEL
LIN {X 0,Y 481.753,Z 96.791,A -85,B 0,C 180,E1 -6761.785,E2 -6761.785} C_VEL
LIN {X 0,Y 481.744,Z 96.786,A -85,B 0,C 180,E1 -6765.225,E2 -6765.225} C_VEL
LIN {X 0,Y 481.714,Z 96.788,A -85,B 0,C 180,E1 -6768.722,E2 -6768.722} C_VEL
LIN {X 0,Y 481.648,Z 96.801,A -85,B 0,C 180,E1 -6771.395,E2 -6771.395} C_VEL
LIN {X 0,Y 481.663,Z 96.797,A -85,B 0,C 180,E1 -6774.114,E2 -6774.114} C_VEL
LIN {X 0,Y 481.749,Z 96.787,A -85,B 0,C 180,E1 -6777.14,E2 -6777.14} C_VEL
LIN {X 0,Y 481.681,Z 96.798,A -85,B 0,C 180,E1 -6779.741,E2 -6779.741} C_VEL
LIN {X 0,Y 481.675,Z 96.793,A -85,B 0,C 180,E1 -6782.675,E2 -6782.675} C_VEL
LIN {X 0,Y 481.639,Z 96.802,A -85,B 0,C 180,E1 -6785.71,E2 -6785.71} C_VEL
LIN {X 0,Y 481.673,Z 96.795,A -85,B 0,C 180,E1 -6788.859,E2 -6788.859} C_VEL
LIN {X 0,Y 481.655,Z 96.797,A -85,B 0,C 180,E1 -6791.913,E2 -6791.913} C_VEL
LIN {X 0,Y 481.662,Z 96.795,A -85,B 0,C 180,E1 -6794.458,E2 -6794.458} C_VEL
LIN {X 0,Y 481.65,Z 96.798,A -85,B 0,C 180,E1 -6797.84,E2 -6797.84} C_VEL
LIN {X 0,Y 481.664,Z 96.797,A -85,B 0,C 180,E1 -6800.654,E2 -6800.654} C_VEL
LIN {X 0,Y 481.631,Z 96.805,A -85,B 0,C 180,E1 -6803.376,E2 -6803.376} C_VEL
LIN {X 0,Y 481.713,Z 96.791,A -85,B 0,C 180,E1 -6806.33,E2 -6806.33} C_VEL
LIN {X 0,Y 481.654,Z 96.801,A -85,B 0,C 180,E1 -6809.418,E2 -6809.418} C_VEL
LIN {X 0,Y 481.742,Z 96.93,A -85,B 0,C 180,E1 -6811.768,E2 -6811.768} C_VEL
LIN {X 0,Y 482.853,Z 99.887,A -85,B 0,C 180,E1 -6811.892,E2 -6811.892} C_VEL
LIN {X 0,Y 492.281,Z 118.943,A -85,B 0,C 180,E1 -6812.801,E2 -6812.801} C_VEL
LIN {X 0,Y 489.585,Z 273.927,A -85,B 0,C 180,E1 -6815.399,E2 -6815.399} C_VEL
LIN {X 0,Y 489.179,Z 295.463,A -85,B 0,C 180,E1 -6815.801,E2 -6815.801} C_VEL
LIN {X 0,Y 488.761,Z 311.529,A -85,B 0,C 180,E1 -6816.258,E2 -6816.258} C_VEL
LIN {X 0,Y 488.148,Z 328.112,A -85,B 0,C 180,E1 -6816.901,E2 -6816.901} C_VEL
LIN {X 0,Y 487.5,Z 343.43,A -85,B 0,C 180,E1 -6817.671,E2 -6817.671} C_VEL
LIN {X 0,Y 486.63,Z 358.725,A -85,B 0,C 180,E1 -6818.613,E2 -6818.613} C_VEL
LIN {X 0,Y 485.817,Z 373.082,A -85,B 0,C 180,E1 -6819.684,E2 -6819.684} C_VEL
LIN {X 0,Y 484.987,Z 386.389,A -85,B 0,C 180,E1 -6820.861,E2 -6820.861} C_VEL
LIN {X 0,Y 484.124,Z 399.644,A -85,B 0,C 180,E1 -6822.25,E2 -6822.25} C_VEL
LIN {X 0,Y 483.334,Z 412.217,A -85,B 0,C 180,E1 -6823.82,E2 -6823.82} C_VEL
LIN {X 0,Y 482.67,Z 423.191,A -85,B 0,C 180,E1 -6825.453,E2 -6825.453} C_VEL
LIN {X 0,Y 482.122,Z 432.785,A -85,B 0,C 180,E1 -6827.156,E2 -6827.156} C_VEL
LIN {X 0,Y 481.776,Z 439.878,A -85,B 0,C 180,E1 -6828.642,E2 -6828.642} C_VEL
LIN {X 0,Y 481.444,Z 446.706,A -85,B 0,C 180,E1 -6830.336,E2 -6830.336} C_VEL
LIN {X 0,Y 481.217,Z 453.428,A -85,B 0,C 180,E1 -6832.447,E2 -6832.447} C_VEL
LIN {X 0,Y 481.062,Z 457.48,A -85,B 0,C 180,E1 -6834.13,E2 -6834.13} C_VEL
LIN {X 0,Y 481,Z 460.543,A -85,B 0,C 180,E1 -6835.81,E2 -6835.81} C_VEL
LIN {X 0,Y 480.939,Z 462.556,A -85,B 0,C 180,E1 -6837.487,E2 -6837.487} C_VEL
LIN {X 0,Y 480.796,Z 463.632,A -85,B 0,C 180,E1 -6839.162,E2 -6839.162} C_VEL
LIN {X 0,Y 480.799,Z 463.716,A -85,B 0,C 180,E1 -6840.837,E2 -6840.837} C_VEL
LIN {X 0,Y 480.94,Z 462.831,A -85,B 0,C 180,E1 -6842.513,E2 -6842.513} C_VEL
LIN {X 0,Y 481.02,Z 460.98,A -85,B 0,C 180,E1 -6844.189,E2 -6844.189} C_VEL
LIN {X 0,Y 481.067,Z 458.099,A -85,B 0,C 180,E1 -6845.869,E2 -6845.869} C_VEL
LIN {X 0,Y 481.255,Z 454.204,A -85,B 0,C 180,E1 -6847.552,E2 -6847.552} C_VEL
LIN {X 0,Y 481.488,Z 447.703,A -85,B 0,C 180,E1 -6849.663,E2 -6849.663} C_VEL
LIN {X 0,Y 481.837,Z 441.044,A -85,B 0,C 180,E1 -6851.356,E2 -6851.356} C_VEL
LIN {X 0,Y 482.254,Z 432.988,A -85,B 0,C 180,E1 -6853.055,E2 -6853.055} C_VEL
LIN {X 0,Y 482.853,Z 423.314,A -85,B 0,C 180,E1 -6854.757,E2 -6854.757} C_VEL
LIN {X 0,Y 483.438,Z 413.646,A -85,B 0,C 180,E1 -6856.202,E2 -6856.202} C_VEL
LIN {X 0,Y 484.236,Z 401.384,A -85,B 0,C 180,E1 -6857.745,E2 -6857.745} C_VEL
LIN {X 0,Y 484.992,Z 388.219,A -85,B 0,C 180,E1 -6859.139,E2 -6859.139} C_VEL
LIN {X 0,Y 485.848,Z 374.97,A -85,B 0,C 180,E1 -6860.314,E2 -6860.314} C_VEL
LIN {X 0,Y 486.621,Z 360.625,A -85,B 0,C 180,E1 -6861.387,E2 -6861.387} C_VEL
LIN {X 0,Y 487.403,Z 345.832,A -85,B 0,C 180,E1 -6862.301,E2 -6862.301} C_VEL
LIN {X 0,Y 488.029,Z 331.08,A -85,B 0,C 180,E1 -6863.049,E2 -6863.049} C_VEL
LIN {X 0,Y 488.576,Z 313.928,A -85,B 0,C 180,E1 -6863.723,E2 -6863.723} C_VEL
LIN {X 0,Y 488.951,Z 297.846,A -85,B 0,C 180,E1 -6864.183,E2 -6864.183} C_VEL
LIN {X 0,Y 489.44,Z 273.137,A -85,B 0,C 180,E1 -6864.647,E2 -6864.647} C_VEL
LIN {X 0,Y 491.375,Z 188.109,A -85,B 0,C 180,E1 -6866.206,E2 -6866.206} C_VEL
LIN {X 0,Y 493.512,Z 119.399,A -85,B 0,C 180,E1 -6867.571,E2 -6867.571} C_VEL
LIN {X 0,Y 486.745,Z 106.52,A -85,B 0,C 180,E1 -6868.425,E2 -6868.425} C_VEL
LIN {X 0,Y 483.356,Z 100.616,A -85,B 0,C 180,E1 -6868.879,E2 -6868.879} C_VEL
LIN {X 0,Y 481.902,Z 98.024,A -85,B 0,C 180,E1 -6869.08,E2 -6869.08} C_VEL
LIN {X 0,Y 481.668,Z 96.8,A -85,B 0,C 180,E1 -6869.159,E2 -6869.159} C_VEL
LIN {X 0,Y 481.671,Z 96.803,A -85,B 0,C 180,E1 -6872.674,E2 -6872.674} C_VEL
LIN {X 0,Y 481.633,Z 96.804,A -85,B 0,C 180,E1 -6875.71,E2 -6875.71} C_VEL
LIN {X 0,Y 481.668,Z 96.801,A -85,B 0,C 180,E1 -6878.859,E2 -6878.859} C_VEL
LIN {X 0,Y 481.654,Z 96.802,A -85,B 0,C 180,E1 -6881.912,E2 -6881.912} C_VEL
LIN {X 0,Y 481.656,Z 96.803,A -85,B 0,C 180,E1 -6884.457,E2 -6884.457} C_VEL
LIN {X 0,Y 481.649,Z 96.804,A -85,B 0,C 180,E1 -6887.839,E2 -6887.839} C_VEL
LIN {X 0,Y 481.681,Z 96.798,A -85,B 0,C 180,E1 -6890.651,E2 -6890.651} C_VEL
LIN {X 0,Y 481.628,Z 96.807,A -85,B 0,C 180,E1 -6893.376,E2 -6893.376} C_VEL
LIN {X 0,Y 481.69,Z 96.874,A -85,B 0,C 180,E1 -6895.317,E2 -6895.317} C_VEL
LIN {X 0,Y 485.746,Z 107.954,A -85,B 0,C 180,E1 -6897.052,E2 -6897.052} C_VEL
LIN {X 0,Y 489.447,Z 120.059,A -85,B 0,C 180,E1 -6898.714,E2 -6898.714} C_VEL
LIN {X 0,Y 490.102,Z 123.293,A -85,B 0,C 180,E1 -6899.105,E2 -6899.105} C_VEL
LIN {X 0,Y 488.536,Z 146.672,A -85,B 0,C 180,E1 -6901.39,E2 -6901.39} C_VEL
LIN {X 0,Y 491.698,Z 169.114,A -85,B 0,C 180,E1 -6902.148,E2 -6902.148} C_VEL
LIN {X 0,Y 492.674,Z 179.097,A -85,B 0,C 180,E1 -6902.436,E2 -6902.436} C_VEL
LIN {X 0,Y 490.038,Z 275.66,A -85,B 0,C 180,E1 -6904.26,E2 -6904.26} C_VEL
LIN {X 0,Y 488.455,Z 360.363,A -85,B 0,C 180,E1 -6905.762,E2 -6905.762} C_VEL
LIN {X 0,Y 487.862,Z 377.093,A -85,B 0,C 180,E1 -6906.211,E2 -6906.211} C_VEL
LIN {X 0,Y 487.113,Z 394.287,A -85,B 0,C 180,E1 -6906.848,E2 -6906.848} C_VEL
LIN {X 0,Y 486.331,Z 409.596,A -85,B 0,C 180,E1 -6907.576,E2 -6907.576} C_VEL
LIN {X 0,Y 485.532,Z 424.656,A -85,B 0,C 180,E1 -6908.45,E2 -6908.45} C_VEL
LIN {X 0,Y 484.717,Z 439.999,A -85,B 0,C 180,E1 -6909.525,E2 -6909.525} C_VEL
LIN {X 0,Y 483.86,Z 454.69,A -85,B 0,C 180,E1 -6910.754,E2 -6910.754} C_VEL
LIN {X 0,Y 483.16,Z 468.273,A -85,B 0,C 180,E1 -6912.104,E2 -6912.104} C_VEL
LIN {X 0,Y 482.556,Z 480.192,A -85,B 0,C 180,E1 -6913.5,E2 -6913.5} C_VEL
LIN {X 0,Y 482.045,Z 491.191,A -85,B 0,C 180,E1 -6915.001,E2 -6915.001} C_VEL
LIN {X 0,Y 481.633,Z 500.628,A -85,B 0,C 180,E1 -6916.498,E2 -6916.498} C_VEL
LIN {X 0,Y 481.347,Z 509.704,A -85,B 0,C 180,E1 -6918.205,E2 -6918.205} C_VEL
LIN {X 0,Y 481.102,Z 517.18,A -85,B 0,C 180,E1 -6919.904,E2 -6919.904} C_VEL
LIN {X 0,Y 481.002,Z 523.343,A -85,B 0,C 180,E1 -6921.598,E2 -6921.598} C_VEL
LIN {X 0,Y 481.009,Z 528.778,A -85,B 0,C 180,E1 -6923.484,E2 -6923.484} C_VEL
LIN {X 0,Y 480.856,Z 531.965,A -85,B 0,C 180,E1 -6924.969,E2 -6924.969} C_VEL
LIN {X 0,Y 480.91,Z 534.661,A -85,B 0,C 180,E1 -6926.648,E2 -6926.648} C_VEL
LIN {X 0,Y 480.824,Z 536.195,A -85,B 0,C 180,E1 -6928.324,E2 -6928.324} C_VEL
LIN {X 0,Y 480.766,Z 536.805,A -85,B 0,C 180,E1 -6929.999,E2 -6929.999} C_VEL
LIN {X 0,Y 480.822,Z 536.301,A -85,B 0,C 180,E1 -6931.675,E2 -6931.675} C_VEL
LIN {X 0,Y 480.891,Z 534.868,A -85,B 0,C 180,E1 -6933.351,E2 -6933.351} C_VEL
LIN {X 0,Y 480.847,Z 532.301,A -85,B 0,C 180,E1 -6935.03,E2 -6935.03} C_VEL
LIN {X 0,Y 480.955,Z 528.734,A -85,B 0,C 180,E1 -6936.713,E2 -6936.713} C_VEL
LIN {X 0,Y 481,Z 523.986,A -85,B 0,C 180,E1 -6938.401,E2 -6938.401} C_VEL
LIN {X 0,Y 481.097,Z 518.029,A -85,B 0,C 180,E1 -6940.095,E2 -6940.095} C_VEL
LIN {X 0,Y 481.357,Z 510.803,A -85,B 0,C 180,E1 -6941.794,E2 -6941.794} C_VEL
LIN {X 0,Y 481.701,Z 502.04,A -85,B 0,C 180,E1 -6943.499,E2 -6943.499} C_VEL
LIN {X 0,Y 482.157,Z 492.958,A -85,B 0,C 180,E1 -6944.994,E2 -6944.994} C_VEL
LIN {X 0,Y 482.704,Z 482.383,A -85,B 0,C 180,E1 -6946.493,E2 -6946.493} C_VEL
LIN {X 0,Y 483.283,Z 471.839,A -85,B 0,C 180,E1 -6947.781,E2 -6947.781} C_VEL
LIN {X 0,Y 484.065,Z 459.039,A -85,B 0,C 180,E1 -6949.121,E2 -6949.121} C_VEL
LIN {X 0,Y 484.924,Z 445.172,A -85,B 0,C 180,E1 -6950.354,E2 -6950.354} C_VEL
LIN {X 0,Y 485.744,Z 430.89,A -85,B 0,C 180,E1 -6951.427,E2 -6951.427} C_VEL
LIN {X 0,Y 486.624,Z 416.688,A -85,B 0,C 180,E1 -6952.317,E2 -6952.317} C_VEL
LIN {X 0,Y 487.483,Z 400.676,A -85,B 0,C 180,E1 -6953.132,E2 -6953.132} C_VEL
LIN {X 0,Y 488.217,Z 384.702,A -85,B 0,C 180,E1 -6953.769,E2 -6953.769} C_VEL
LIN {X 0,Y 488.82,Z 368.781,A -85,B 0,C 180,E1 -6954.245,E2 -6954.245} C_VEL
LIN {X 0,Y 489.306,Z 351.978,A -85,B 0,C 180,E1 -6954.587,E2 -6954.587} C_VEL
LIN {X 0,Y 492.26,Z 178.053,A -85,B 0,C 180,E1 -6957.494,E2 -6957.494} C_VEL
LIN {X 0,Y 488.608,Z 153.572,A -85,B 0,C 180,E1 -6958.161,E2 -6958.161} C_VEL
LIN {X 0,Y 490.16,Z 123.684,A -85,B 0,C 180,E1 -6960.912,E2 -6960.912} C_VEL
LIN {X 0,Y 485.095,Z 107.248,A -85,B 0,C 180,E1 -6962.829,E2 -6962.829} C_VEL
LIN {X 0,Y 481.703,Z 96.795,A -85,B 0,C 180,E1 -6964.108,E2 -6964.108} C_VEL
LIN {X 0,Y 481.621,Z 96.808,A -85,B 0,C 180,E1 -6966.747,E2 -6966.747} C_VEL
LIN {X 0,Y 481.672,Z 96.799,A -85,B 0,C 180,E1 -6969.94,E2 -6969.94} C_VEL
LIN {X 0,Y 481.68,Z 96.794,A -85,B 0,C 180,E1 -6973.294,E2 -6973.294} C_VEL
LIN {X 0,Y 481.634,Z 96.802,A -85,B 0,C 180,E1 -6976.7,E2 -6976.7} C_VEL
LIN {X 0,Y 481.672,Z 96.798,A -85,B 0,C 180,E1 -6980.059,E2 -6980.059} C_VEL
LIN {X 0,Y 481.625,Z 96.799,A -85,B 0,C 180,E1 -6983.253,E2 -6983.253} C_VEL
LIN {X 0,Y 481.705,Z 96.796,A -85,B 0,C 180,E1 -6986.33,E2 -6986.33} C_VEL
LIN {X 0,Y 481.647,Z 96.797,A -85,B 0,C 180,E1 -6989.417,E2 -6989.417} C_VEL
LIN {X 0,Y 481.696,Z 96.798,A -85,B 0,C 180,E1 -6992.168,E2 -6992.168} C_VEL
LIN {X 0,Y 481.714,Z 96.788,A -85,B 0,C 180,E1 -6994.97,E2 -6994.97} C_VEL
LIN {X 0,Y 481.648,Z 96.801,A -85,B 0,C 180,E1 -6997.705,E2 -6997.705} C_VEL
LIN {X 0,Y 481.701,Z 96.793,A -85,B 0,C 180,E1 -7000.393,E2 -7000.393} C_VEL
LIN {X 0,Y 481.686,Z 96.792,A -85,B 0,C 180,E1 -7003.034,E2 -7003.034} C_VEL
LIN {X 0,Y 481.686,Z 96.797,A -85,B 0,C 180,E1 -7005.639,E2 -7005.639} C_VEL
LIN {X 0,Y 481.791,Z 96.782,A -85,B 0,C 180,E1 -7008.216,E2 -7008.216} C_VEL
LIN {X 0,Y 481.758,Z 96.789,A -85,B 0,C 180,E1 -7011.612,E2 -7011.612} C_VEL
LIN {X 0,Y 481.811,Z 96.779,A -85,B 0,C 180,E1 -7014.14,E2 -7014.14} C_VEL
LIN {X 0,Y 481.923,Z 96.768,A -85,B 0,C 180,E1 -7017.493,E2 -7017.493} C_VEL
LIN {X 0,Y 481.901,Z 96.765,A -85,B 0,C 180,E1 -7020.836,E2 -7020.836} C_VEL
LIN {X 0,Y 481.924,Z 96.762,A -85,B 0,C 180,E1 -7022.508,E2 -7022.508} C_VEL
LIN {X 0,Y 481.812,Z 96.78,A -85,B 0,C 180,E1 -7025.861,E2 -7025.861} C_VEL
LIN {X 0,Y 481.758,Z 96.783,A -85,B 0,C 180,E1 -7028.388,E2 -7028.388} C_VEL
LIN {X 0,Y 481.746,Z 96.788,A -85,B 0,C 180,E1 -7031.785,E2 -7031.785} C_VEL
LIN {X 0,Y 481.738,Z 96.792,A -85,B 0,C 180,E1 -7035.224,E2 -7035.224} C_VEL
LIN {X 0,Y 481.708,Z 96.791,A -85,B 0,C 180,E1 -7038.722,E2 -7038.722} C_VEL
LIN {X 0,Y 481.643,Z 96.804,A -85,B 0,C 180,E1 -7041.395,E2 -7041.395} C_VEL
LIN {X 0,Y 481.673,Z 96.793,A -85,B 0,C 180,E1 -7044.113,E2 -7044.113} C_VEL
LIN {X 0,Y 481.743,Z 96.793,A -85,B 0,C 180,E1 -7047.14,E2 -7047.14} C_VEL
LIN {X 0,Y 481.675,Z 96.794,A -85,B 0,C 180,E1 -7049.741,E2 -7049.741} C_VEL
LIN {X 0,Y 481.669,Z 96.797,A -85,B 0,C 180,E1 -7052.674,E2 -7052.674} C_VEL
LIN {X 0,Y 481.639,Z 96.798,A -85,B 0,C 180,E1 -7055.709,E2 -7055.709} C_VEL
LIN {X 0,Y 481.668,Z 96.801,A -85,B 0,C 180,E1 -7058.859,E2 -7058.859} C_VEL
LIN {X 0,Y 481.659,Z 96.795,A -85,B 0,C 180,E1 -7061.915,E2 -7061.915} C_VEL
LIN {X 0,Y 481.657,Z 96.799,A -85,B 0,C 180,E1 -7064.458,E2 -7064.458} C_VEL
LIN {X 0,Y 481.651,Z 96.796,A -85,B 0,C 180,E1 -7067.841,E2 -7067.841} C_VEL
LIN {X 0,Y 481.701,Z 96.797,A -85,B 0,C 180,E1 -7070.648,E2 -7070.648} C_VEL
LIN {X 0,Y 481.624,Z 96.8,A -85,B 0,C 180,E1 -7073.377,E2 -7073.377} C_VEL
LIN {X 0,Y 481.707,Z 96.793,A -85,B 0,C 180,E1 -7076.331,E2 -7076.331} C_VEL
LIN {X 0,Y 481.648,Z 96.797,A -85,B 0,C 180,E1 -7079.418,E2 -7079.418} C_VEL
LIN {X 0,Y 481.698,Z 96.794,A -85,B 0,C 180,E1 -7082.169,E2 -7082.169} C_VEL
LIN {X 0,Y 481.717,Z 96.79,A -85,B 0,C 180,E1 -7084.971,E2 -7084.971} C_VEL
LIN {X 0,Y 481.635,Z 96.799,A -85,B 0,C 180,E1 -7087.983,E2 -7087.983} C_VEL
LIN {X 0,Y 480.967,Z 96.887,A -85,B 0,C 180,E1 -7088.681,E2 -7088.681} C_VEL
LIN {X 0,Y 478.14,Z 97.235,A -85,B 0,C 180,E1 -7089.815,E2 -7089.815} C_VEL
LIN {X 0,Y 475.756,Z 97.534,A -85,B 0,C 180,E1 -7090.729,E2 -7090.729} C_VEL
LIN {X 0,Y 474.736,Z 97.658,A -85,B 0,C 180,E1 -7091.435,E2 -7091.435} C_VEL
LIN {X 0,Y 474.655,Z 97.668,A -85,B 0,C 180,E1 -7091.674,E2 -7091.674} C_VEL
LIN {X 0,Y 474.699,Z 97.667,A -85,B 0,C 180,E1 -7094.545,E2 -7094.545} C_VEL
LIN {X 0,Y 474.704,Z 97.667,A -85,B 0,C 180,E1 -7098.038,E2 -7098.038} C_VEL
LIN {X 0,Y 474.728,Z 97.659,A -85,B 0,C 180,E1 -7101.487,E2 -7101.487} C_VEL
LIN {X 0,Y 474.779,Z 97.659,A -85,B 0,C 180,E1 -7104.053,E2 -7104.053} C_VEL
LIN {X 0,Y 474.894,Z 97.639,A -85,B 0,C 180,E1 -7107.456,E2 -7107.456} C_VEL
LIN {X 0,Y 474.912,Z 97.643,A -85,B 0,C 180,E1 -7110.001,E2 -7110.001} C_VEL
LIN {X 0,Y 474.894,Z 97.64,A -85,B 0,C 180,E1 -7112.545,E2 -7112.545} C_VEL
LIN {X 0,Y 474.779,Z 97.661,A -85,B 0,C 180,E1 -7115.948,E2 -7115.948} C_VEL
LIN {X 0,Y 474.729,Z 97.66,A -85,B 0,C 180,E1 -7118.514,E2 -7118.514} C_VEL
LIN {X 0,Y 474.706,Z 97.668,A -85,B 0,C 180,E1 -7121.963,E2 -7121.963} C_VEL
LIN {X 0,Y 474.702,Z 97.666,A -85,B 0,C 180,E1 -7125.456,E2 -7125.456} C_VEL
LIN {X 0,Y 474.667,Z 97.667,A -85,B 0,C 180,E1 -7129.011,E2 -7129.011} C_VEL
LIN {X 0,Y 474.591,Z 97.683,A -85,B 0,C 180,E1 -7131.729,E2 -7131.729} C_VEL
LIN {X 0,Y 474.643,Z 97.669,A -85,B 0,C 180,E1 -7134.494,E2 -7134.494} C_VEL
LIN {X 0,Y 474.702,Z 97.667,A -85,B 0,C 180,E1 -7137.339,E2 -7137.339} C_VEL
LIN {X 0,Y 474.607,Z 97.674,A -85,B 0,C 180,E1 -7140.811,E2 -7140.811} C_VEL
LIN {X 0,Y 474.64,Z 97.672,A -85,B 0,C 180,E1 -7143.984,E2 -7143.984} C_VEL
LIN {X 0,Y 474.574,Z 97.68,A -85,B 0,C 180,E1 -7146.9,E2 -7146.9} C_VEL
LIN {X 0,Y 474.63,Z 97.675,A -85,B 0,C 180,E1 -7149.648,E2 -7149.648} C_VEL
LIN {X 0,Y 474.618,Z 97.676,A -85,B 0,C 180,E1 -7152.935,E2 -7152.935} C_VEL
LIN {X 0,Y 474.612,Z 97.674,A -85,B 0,C 180,E1 -7155.895,E2 -7155.895} C_VEL
LIN {X 0,Y 474.63,Z 97.677,A -85,B 0,C 180,E1 -7159.041,E2 -7159.041} C_VEL
LIN {X 0,Y 474.613,Z 97.675,A -85,B 0,C 180,E1 -7161.704,E2 -7161.704} C_VEL
LIN {X 0,Y 474.63,Z 97.677,A -85,B 0,C 180,E1 -7164.726,E2 -7164.726} C_VEL
LIN {X 0,Y 474.639,Z 97.674,A -85,B 0,C 180,E1 -7167.788,E2 -7167.788} C_VEL
LIN {X 0,Y 474.689,Z 97.827,A -85,B 0,C 180,E1 -7171.352,E2 -7171.352} C_VEL
LIN {X 0,Y 475.814,Z 100.748,A -85,B 0,C 180,E1 -7171.479,E2 -7171.479} C_VEL
LIN {X 0,Y 485.869,Z 120.948,A -85,B 0,C 180,E1 -7172.468,E2 -7172.468} C_VEL
LIN {X 0,Y 482.994,Z 274.806,A -85,B 0,C 180,E1 -7175.098,E2 -7175.098} C_VEL
LIN {X 0,Y 482.581,Z 296.103,A -85,B 0,C 180,E1 -7175.506,E2 -7175.506} C_VEL
LIN {X 0,Y 482.088,Z 312.83,A -85,B 0,C 180,E1 -7175.994,E2 -7175.994} C_VEL
LIN {X 0,Y 481.496,Z 328.634,A -85,B 0,C 180,E1 -7176.62,E2 -7176.62} C_VEL
LIN {X 0,Y 480.839,Z 343.513,A -85,B 0,C 180,E1 -7177.378,E2 -7177.378} C_VEL
LIN {X 0,Y 479.949,Z 358.416,A -85,B 0,C 180,E1 -7178.3,E2 -7178.3} C_VEL
LIN {X 0,Y 479.049,Z 372.914,A -85,B 0,C 180,E1 -7179.384,E2 -7179.384} C_VEL
LIN {X 0,Y 478.199,Z 386.338,A -85,B 0,C 180,E1 -7180.578,E2 -7180.578} C_VEL
LIN {X 0,Y 477.282,Z 399.702,A -85,B 0,C 180,E1 -7181.987,E2 -7181.987} C_VEL
LIN {X 0,Y 476.531,Z 411.483,A -85,B 0,C 180,E1 -7183.465,E2 -7183.465} C_VEL
LIN {X 0,Y 475.828,Z 422.04,A -85,B 0,C 180,E1 -7185.02,E2 -7185.02} C_VEL
LIN {X 0,Y 475.226,Z 431.954,A -85,B 0,C 180,E1 -7186.748,E2 -7186.748} C_VEL
LIN {X 0,Y 474.767,Z 440.229,A -85,B 0,C 180,E1 -7188.472,E2 -7188.472} C_VEL
LIN {X 0,Y 474.405,Z 447.095,A -85,B 0,C 180,E1 -7190.191,E2 -7190.191} C_VEL
LIN {X 0,Y 474.165,Z 453.866,A -85,B 0,C 180,E1 -7192.334,E2 -7192.334} C_VEL
LIN {X 0,Y 474.015,Z 457.947,A -85,B 0,C 180,E1 -7194.043,E2 -7194.043} C_VEL
LIN {X 0,Y 473.941,Z 461.04,A -85,B 0,C 180,E1 -7195.748,E2 -7195.748} C_VEL
LIN {X 0,Y 473.883,Z 463.072,A -85,B 0,C 180,E1 -7197.45,E2 -7197.45} C_VEL
LIN {X 0,Y 473.722,Z 464.167,A -85,B 0,C 180,E1 -7199.15,E2 -7199.15} C_VEL
LIN {X 0,Y 473.725,Z 464.263,A -85,B 0,C 180,E1 -7200.85,E2 -7200.85} C_VEL
LIN {X 0,Y 473.885,Z 463.38,A -85,B 0,C 180,E1 -7202.55,E2 -7202.55} C_VEL
LIN {X 0,Y 473.962,Z 461.533,A -85,B 0,C 180,E1 -7204.252,E2 -7204.252} C_VEL
LIN {X 0,Y 474.021,Z 458.649,A -85,B 0,C 180,E1 -7205.957,E2 -7205.957} C_VEL
LIN {X 0,Y 474.229,Z 454.751,A -85,B 0,C 180,E1 -7207.665,E2 -7207.665} C_VEL
LIN {X 0,Y 474.478,Z 448.23,A -85,B 0,C 180,E1 -7209.807,E2 -7209.807} C_VEL
LIN {X 0,Y 474.861,Z 441.562,A -85,B 0,C 180,E1 -7211.525,E2 -7211.525} C_VEL
LIN {X 0,Y 475.305,Z 433.491,A -85,B 0,C 180,E1 -7213.249,E2 -7213.249} C_VEL
LIN {X 0,Y 475.974,Z 423.784,A -85,B 0,C 180,E1 -7214.975,E2 -7214.975} C_VEL
LIN {X 0,Y 476.567,Z 414.482,A -85,B 0,C 180,E1 -7216.388,E2 -7216.388} C_VEL
LIN {X 0,Y 477.46,Z 401.81,A -85,B 0,C 180,E1 -7218.006,E2 -7218.006} C_VEL
LIN {X 0,Y 478.264,Z 388.623,A -85,B 0,C 180,E1 -7219.419,E2 -7219.419} C_VEL
LIN {X 0,Y 479.24,Z 374.047,A -85,B 0,C 180,E1 -7220.719,E2 -7220.719} C_VEL
LIN {X 0,Y 480.079,Z 359.379,A -85,B 0,C 180,E1 -7221.806,E2 -7221.806} C_VEL
LIN {X 0,Y 480.891,Z 344.584,A -85,B 0,C 180,E1 -7222.708,E2 -7222.708} C_VEL
LIN {X 0,Y 481.558,Z 328.774,A -85,B 0,C 180,E1 -7223.491,E2 -7223.491} C_VEL
LIN {X 0,Y 482.152,Z 312.403,A -85,B 0,C 180,E1 -7224.116,E2 -7224.116} C_VEL
LIN {X 0,Y 482.537,Z 297.04,A -85,B 0,C 180,E1 -7224.554,E2 -7224.554} C_VEL
LIN {X 0,Y 484.919,Z 197.468,A -85,B 0,C 180,E1 -7226.437,E2 -7226.437} C_VEL
LIN {X 0,Y 487.626,Z 122.354,A -85,B 0,C 180,E1 -7227.967,E2 -7227.967} C_VEL
LIN {X 0,Y 482.812,Z 112.506,A -85,B 0,C 180,E1 -7228.617,E2 -7228.617} C_VEL
LIN {X 0,Y 477.947,Z 104.248,A -85,B 0,C 180,E1 -7229.288,E2 -7229.288} C_VEL
LIN {X 0,Y 476.441,Z 101.572,A -85,B 0,C 180,E1 -7229.504,E2 -7229.504} C_VEL
LIN {X 0,Y 474.91,Z 98.958,A -85,B 0,C 180,E1 -7229.733,E2 -7229.733} C_VEL
LIN {X 0,Y 474.623,Z 97.679,A -85,B 0,C 180,E1 -7229.805,E2 -7229.805} C_VEL
LIN {X 0,Y 474.626,Z 97.679,A -85,B 0,C 180,E1 -7233.221,E2 -7233.221} C_VEL
LIN {X 0,Y 474.586,Z 97.684,A -85,B 0,C 180,E1 -7236.324,E2 -7236.324} C_VEL
LIN {X 0,Y 474.617,Z 97.678,A -85,B 0,C 180,E1 -7239.645,E2 -7239.645} C_VEL
LIN {X 0,Y 474.626,Z 97.678,A -85,B 0,C 180,E1 -7242.236,E2 -7242.236} C_VEL
LIN {X 0,Y 474.618,Z 97.677,A -85,B 0,C 180,E1 -7245.297,E2 -7245.297} C_VEL
LIN {X 0,Y 474.622,Z 97.68,A -85,B 0,C 180,E1 -7248.214,E2 -7248.214} C_VEL
LIN {X 0,Y 474.646,Z 97.676,A -85,B 0,C 180,E1 -7250.454,E2 -7250.454} C_VEL
LIN {X 0,Y 474.59,Z 97.685,A -85,B 0,C 180,E1 -7253.676,E2 -7253.676} C_VEL
LIN {X 0,Y 474.645,Z 97.879,A -85,B 0,C 180,E1 -7254.638,E2 -7254.638} C_VEL
LIN {X 0,Y 479.317,Z 110.123,A -85,B 0,C 180,E1 -7256.695,E2 -7256.695} C_VEL
LIN {X 0,Y 482.96,Z 122.177,A -85,B 0,C 180,E1 -7258.407,E2 -7258.407} C_VEL
LIN {X 0,Y 483.705,Z 125.867,A -85,B 0,C 180,E1 -7258.874,E2 -7258.874} C_VEL
LIN {X 0,Y 482.234,Z 145.701,A -85,B 0,C 180,E1 -7260.856,E2 -7260.856} C_VEL
LIN {X 0,Y 485.501,Z 168.909,A -85,B 0,C 180,E1 -7261.682,E2 -7261.682} C_VEL
LIN {X 0,Y 486.602,Z 179.808,A -85,B 0,C 180,E1 -7262.018,E2 -7262.018} C_VEL
LIN {X 0,Y 483.759,Z 273.133,A -85,B 0,C 180,E1 -7263.843,E2 -7263.843} C_VEL
LIN {X 0,Y 481.894,Z 360.066,A -85,B 0,C 180,E1 -7265.439,E2 -7265.439} C_VEL
LIN {X 0,Y 481.23,Z 377.335,A -85,B 0,C 180,E1 -7265.92,E2 -7265.92} C_VEL
LIN {X 0,Y 480.417,Z 394.263,A -85,B 0,C 180,E1 -7266.563,E2 -7266.563} C_VEL
LIN {X 0,Y 479.528,Z 410.782,A -85,B 0,C 180,E1 -7267.375,E2 -7267.375} C_VEL
LIN {X 0,Y 478.588,Z 426.784,A -85,B 0,C 180,E1 -7268.348,E2 -7268.348} C_VEL
LIN {X 0,Y 477.722,Z 441.603,A -85,B 0,C 180,E1 -7269.437,E2 -7269.437} C_VEL
LIN {X 0,Y 476.81,Z 456.322,A -85,B 0,C 180,E1 -7270.722,E2 -7270.722} C_VEL
LIN {X 0,Y 476.164,Z 468.279,A -85,B 0,C 180,E1 -7271.943,E2 -7271.943} C_VEL
LIN {X 0,Y 475.495,Z 481,A -85,B 0,C 180,E1 -7273.469,E2 -7273.469} C_VEL
LIN {X 0,Y 474.97,Z 491.771,A -85,B 0,C 180,E1 -7274.992,E2 -7274.992} C_VEL
LIN {X 0,Y 474.511,Z 502.215,A -85,B 0,C 180,E1 -7276.728,E2 -7276.728} C_VEL
LIN {X 0,Y 474.219,Z 510.945,A -85,B 0,C 180,E1 -7278.458,E2 -7278.458} C_VEL
LIN {X 0,Y 473.985,Z 518.191,A -85,B 0,C 180,E1 -7280.182,E2 -7280.182} C_VEL
LIN {X 0,Y 473.914,Z 524.018,A -85,B 0,C 180,E1 -7281.901,E2 -7281.901} C_VEL
LIN {X 0,Y 473.928,Z 528.4,A -85,B 0,C 180,E1 -7283.491,E2 -7283.491} C_VEL
LIN {X 0,Y 473.806,Z 532.869,A -85,B 0,C 180,E1 -7285.746,E2 -7285.746} C_VEL
LIN {X 0,Y 473.864,Z 534.999,A -85,B 0,C 180,E1 -7287.449,E2 -7287.449} C_VEL
LIN {X 0,Y 473.702,Z 536.078,A -85,B 0,C 180,E1 -7289.149,E2 -7289.149} C_VEL
LIN {X 0,Y 473.699,Z 536.142,A -85,B 0,C 180,E1 -7290.85,E2 -7290.85} C_VEL
